	{attribute 'TcIecLibraryType'}
	{attribute 'external_name' := 'F_VN_SeparableCustomFilter_GUID_FC6321D5_149B_44BA_FE2A_AFF910B64319'}
	(* Apply a separable custom filter to the image. *)
	FUNCTION F_VN_SeparableCustomFilter : HRESULT
	VAR_INPUT
		ipSrcImage	:	ITcVnImage;	(* Source image *)
		ipDestImage	:	REFERENCE TO ITcVnImage;	(* Destination image (An appropriate destination image will be created if required.) *)
		eDestDepth	:	ETcVnElementType;	(* Destination image depth *)
	END_VAR
	VAR_IN_OUT
		stKernelX	:	TcVnMatrix;	(* 1D custom row-filter kernel with values of type REAL or LREAL *)
		stKernelY	:	TcVnMatrix;	(* 1D custom column-filter kernel with values of type REAL or LREAL *)
	END_VAR
	VAR_INPUT
		hrPrev	:	HRESULT;	(* HRESULT indicating the result of previous operations (If SUCCEEDED(hrPrev) equals false, no operation is executed.) *)
	END_VAR

END_FUNCTION

// Functions/Image Filtering/F_VN_SeparableCustomFilterExp

	{attribute 'TcIecLibraryType'}
	{attribute 'external_name' := 'F_VN_SeparableCustomFilterExp_GUID_53B70F4F_154A_462E_D532_DBD6B183CFE7'}
	(* Apply a separable custom filter to the image. (expert function) *)
	FUNCTION F_VN_SeparableCustomFilterExp : HRESULT
	VAR_INPUT
		ipSrcImage	:	ITcVnImage;	(* Source image *)
		ipDestImage	:	REFERENCE TO ITcVnImage;	(* Destination image (An appropriate destination image will be created if required.) *)
		eDestDepth	:	ETcVnElementType;	(* Destination image depth *)
	END_VAR
	VAR_IN_OUT
		stKernelX	:	TcVnMatrix;	(* 1D custom row-filter kernel with values of type REAL or LREAL *)
		stKernelY	:	TcVnMatrix;	(* 1D custom column-filter kernel with values of type REAL or LREAL *)
		aAnchor	:	TcVnPoint;	(* Anchor point of the kernel *)
	END_VAR
	VAR_INPUT
		fDelta	:	LREAL;	(* Value added to each pixel after filtering *)
		eBorderType	:	ETcVnBorderInterpolationMethod;	(* Image border handling *)
		hrPrev	:	HRESULT;	(* HRESULT indicating the result of previous operations (If SUCCEEDED(hrPrev) equals false, no operation is executed.) *)
	END_VAR

END_FUNCTION

// Functions/Image Filtering/F_VN_SobelFilter

	{attribute 'TcIecLibraryType'}
	{attribute 'external_name' := 'F_VN_SobelFilter_GUID_E75A9F88_EB52_4C01_DC1F_4C53F4C1A62C'}
	(* Calculates the first, second, or mixed image derivatives using an extended Sobel filter. *)
	FUNCTION F_VN_SobelFilter : HRESULT
	VAR_INPUT
		ipSrcImage	:	ITcVnImage;	(* Source image *)
		ipDestImage	:	REFERENCE TO ITcVnImage;	(* Destination image (An appropriate destination image will be created if required.) *)
		eDestDepth	:	ETcVnElementType;	(* Destination image depth *)
		nXOrder	:	UDINT;	(* Order of the x-derivative (0, 1, 2) *)
		nYOrder	:	UDINT;	(* Order of the y-derivative (0, 1, 2) *)
		hrPrev	:	HRESULT;	(* HRESULT indicating the result of previous operations (If SUCCEEDED(hrPrev) equals false, no operation is executed.) *)
	END_VAR

END_FUNCTION

// Functions/Image Filtering/F_VN_SobelFilterExp

	{attribute 'TcIecLibraryType'}
	{attribute 'external_name' := 'F_VN_SobelFilterExp_GUID_6432B4D4_802B_419E_F701_7BF4156B289B'}
	(* Calculates the first, second, third, or mixed image derivatives using an extended Sobel filter. (expert function) *)
	FUNCTION F_VN_SobelFilterExp : HRESULT
	VAR_INPUT
		ipSrcImage	:	ITcVnImage;	(* Source image *)
		ipDestImage	:	REFERENCE TO ITcVnImage;	(* Destination image (An appropriate destination image will be created if required.) *)
		eDestDepth	:	ETcVnElementType;	(* Destination image depth *)
		nXOrder	:	UDINT;	(* Order of the x-derivative (must be < nKernelSize) *)
		nYOrder	:	UDINT;	(* Order of the y-derivative (must be < nKernelSize) *)
		nKernelSize	:	UDINT;	(* Size of the extended Sobel kernel (3, 5, 7, ..., 31) *)
		fScale	:	LREAL;	(* Scale factor for the computed derivative values *)
		fDelta	:	LREAL;	(* Delta value that is added to the results prior to storing them in dest *)
		eBorderType	:	ETcVnBorderInterpolationMethod;	(* Image border handling *)
		hrPrev	:	HRESULT;	(* HRESULT indicating the result of previous operations (If SUCCEEDED(hrPrev) equals false, no operation is executed.) *)
	END_VAR

END_FUNCTION

// Functions/Image Filtering/F_VN_VarianceFilter

	{attribute 'TcIecLibraryType'}
	{attribute 'external_name' := 'F_VN_VarianceFilter_GUID_EDB0D6CF_7F73_4B27_CF92_1DD3947C3E57'}
	(* Calculates the local variance of an image. *)
	FUNCTION F_VN_VarianceFilter : HRESULT
	VAR_INPUT
		ipSrcImage	:	ITcVnImage;	(* Source image. Only TCVN_ET_USINT Type is supported.  *)
		ipDestImage	:	REFERENCE TO ITcVnImage;	(* Destination image of type TCVN_ET_UINT (An appropriate destination image will be created if required.) *)
		nKernelSize	:	UDINT;	(* Size of the kernel *)
		hrPrev	:	HRESULT;	(* HRESULT indicating the result of previous operations (If SUCCEEDED(hrPrev) equals false, no operation is executed.) *)
	END_VAR

END_FUNCTION

// Functions/Image Filtering/F_VN_VarianceFilterExp

	{attribute 'TcIecLibraryType'}
	{attribute 'external_name' := 'F_VN_VarianceFilterExp_GUID_A7B8D649_AD30_4302_EB39_E9340C7CCFE8'}
	(* Calculates the local variance of an image. (expert function) *)
	FUNCTION F_VN_VarianceFilterExp : HRESULT
	VAR_INPUT
		ipSrcImage	:	ITcVnImage;	(* Source image. Only TCVN_ET_USINT Type is supported. *)
		ipDestImage	:	REFERENCE TO ITcVnImage;	(* Destination image of type TCVN_ET_UINT (An appropriate destination image will be created if required.) *)
		nKernelSize	:	UDINT;	(* Size of the kernel *)
		fScale	:	LREAL;	(* Scale factor for the computed variance values *)
		eBorderType	:	ETcVnBorderInterpolationMethod;	(* Image border handling *)
		hrPrev	:	HRESULT;	(* HRESULT indicating the result of previous operations (If SUCCEEDED(hrPrev) equals false, no operation is executed.) *)
	END_VAR

END_FUNCTION

// Functions/Miscellaneous/F_VN_CheckFunctionInitialization

	{attribute 'TcIecLibraryType'}
	{attribute 'external_name' := 'F_VN_CheckFunctionInitialization_GUID_C3F1DDC0_B6F9_4195_C99F_AF034AC9584D'}
	(* Check if a function is initialized with the specified options. *)
	FUNCTION F_VN_CheckFunctionInitialization : HRESULT
	VAR_INPUT
		eFunction	:	ETcVnInitializableFunction;	(* Initializable function *)
		nOptions	:	ULINT;	(* Initialization options for the function *)
		hrPrev	:	HRESULT;	(* HRESULT indicating the result of previous operations (If SUCCEEDED(hrPrev) equals false, no operation is executed.) *)
	END_VAR

END_FUNCTION

// Functions/Miscellaneous/F_VN_ClipLineToBoundary

	{attribute 'TcIecLibraryType'}
	{attribute 'external_name' := 'F_VN_ClipLineToBoundary_GUID_5BF147CC_4437_4411_DA65_9BE106D06E3D'}
	(* Clips a line to a rectangular boundary. *)
	FUNCTION F_VN_ClipLineToBoundary : HRESULT
	VAR_IN_OUT
		aLine	:	TcVnVector4_LREAL;	(* The first and second element describe the x and y component of the direction vector. The third and fourth element describe the x and y component of the position vector. *)
	END_VAR
	VAR_INPUT
		nX1	:	DINT;	(* x of top left rectangle point *)
		nY1	:	DINT;	(* y of top left rectangle point *)
		nX2	:	DINT;	(* x of bottom right rectangle point *)
		nY2	:	DINT;	(* Y of bottom right rectangle point *)
	END_VAR
	VAR_IN_OUT
		aStartPoint	:	TcVnPoint2_REAL;	(* Returns the clipped starting point of the line. *)
		aEndPoint	:	TcVnPoint2_REAL;	(* Returns the clipped end point of the line. *)
	END_VAR
	VAR_INPUT
		hrPrev	:	HRESULT;	(* HRESULT indicating the result of previous operations (If SUCCEEDED(hrPrev) equals false, no operation is executed.) *)
	END_VAR

END_FUNCTION

// Functions/Miscellaneous/F_VN_ClipLineToBoundary_ITcVnImage

	{attribute 'TcIecLibraryType'}
	{attribute 'external_name' := 'F_VN_ClipLineToBoundary_ITcVnImage_GUID_E0B9D53C_4691_4392_C0F0_296578E237CB'}
	(* Clips a line to the boundary of an image. *)
	FUNCTION F_VN_ClipLineToBoundary_ITcVnImage : HRESULT
	VAR_IN_OUT
		aLine	:	TcVnVector4_LREAL;	(* The first and second element describe the x and y component of the direction vector. The third and fourth element describe the x and y component of the position vector. *)
	END_VAR
	VAR_INPUT
		ipImage	:	ITcVnImage;	(* Image, from which to derive the boundary *)
	END_VAR
	VAR_IN_OUT
		aStartPoint	:	TcVnPoint2_REAL;	(* Returns the clipped starting point of the line. *)
		aEndPoint	:	TcVnPoint2_REAL;	(* Returns the clipped end point of the line. *)
	END_VAR
	VAR_INPUT
		hrPrev	:	HRESULT;	(* HRESULT indicating the result of previous operations (If SUCCEEDED(hrPrev) equals false, no operation is executed.) *)
	END_VAR

END_FUNCTION

// Functions/Miscellaneous/F_VN_ClipLineToBoundary_TcVnRectangle_DINT

	{attribute 'TcIecLibraryType'}
	{attribute 'external_name' := 'F_VN_ClipLineToBoundary_TcVnRectangle_DINT_GUID_83796845_DAE2_42E1_D405_180DCCA547A8'}
	(* Clips a line to a rectangular boundary. *)
	FUNCTION F_VN_ClipLineToBoundary_TcVnRectangle_DINT : HRESULT
	VAR_IN_OUT
		aLine	:	TcVnVector4_LREAL;	(* The first and second element describe the x and y component of the direction vector. The third and fourth element describe the x and y component of the position vector. *)
		stRectangle	:	TcVnRectangle_DINT;	(* Rectangular boundary *)
		aStartPoint	:	TcVnPoint2_REAL;	(* Returns the clipped starting point of the line. *)
		aEndPoint	:	TcVnPoint2_REAL;	(* Returns the clipped end point of the line. *)
	END_VAR
	VAR_INPUT
		hrPrev	:	HRESULT;	(* HRESULT indicating the result of previous operations (If SUCCEEDED(hrPrev) equals false, no operation is executed.) *)
	END_VAR

END_FUNCTION

// Functions/Miscellaneous/F_VN_ConvertITcUnknownToITcVnBitmapExport

	{attribute 'TcIecLibraryType'}
	{attribute 'external_name' := 'F_VN_ConvertITcUnknownToITcVnBitmapExport_GUID_2ADFAF32_D897_4264_C580_D49D5C531DA7'}
	(* Convert an ITcUnknown interface pointer to an ITcVnBitmapExport interface pointer. The destination pointer will be released (if existing) and set to the source pointer. The source pointer will be set to 0. *)
	FUNCTION F_VN_ConvertITcUnknownToITcVnBitmapExport : HRESULT
	VAR_INPUT
		ipSrc	:	REFERENCE TO ITcUnknown;	(* Source pointer *)
		ipDest	:	REFERENCE TO ITcVnBitmapExport;	(* Destination pointer *)
		hrPrev	:	HRESULT;	(* HRESULT indicating the result of previous operations (If SUCCEEDED(hrPrev) equals false, no operation is executed.) *)
	END_VAR

END_FUNCTION

// Functions/Miscellaneous/F_VN_ConvertITcUnknownToITcVnContainer

	{attribute 'TcIecLibraryType'}
	{attribute 'external_name' := 'F_VN_ConvertITcUnknownToITcVnContainer_GUID_17E3F6C3_BFE3_44EF_FE9F_96A9CAE713C6'}
	(* Convert an ITcUnknown interface pointer to an ITcVnContainer interface pointer. The destination pointer will be released (if existing) and set to the source pointer. The source pointer will be set to 0. *)
	FUNCTION F_VN_ConvertITcUnknownToITcVnContainer : HRESULT
	VAR_INPUT
		ipSrc	:	REFERENCE TO ITcUnknown;	(* Source pointer *)
		ipDest	:	REFERENCE TO ITcVnContainer;	(* Destination pointer *)
		hrPrev	:	HRESULT;	(* HRESULT indicating the result of previous operations (If SUCCEEDED(hrPrev) equals false, no operation is executed.) *)
	END_VAR

END_FUNCTION

// Functions/Miscellaneous/F_VN_ConvertITcUnknownToITcVnImage

	{attribute 'TcIecLibraryType'}
	{attribute 'external_name' := 'F_VN_ConvertITcUnknownToITcVnImage_GUID_181BB9EC_9169_4CB5_D135_A350734A00A3'}
	(* Convert an ITcUnknown interface pointer to an ITcVnImage interface pointer. The destination pointer will be released (if existing) and set to the source pointer. The source pointer will be set to 0. *)
	FUNCTION F_VN_ConvertITcUnknownToITcVnImage : HRESULT
	VAR_INPUT
		ipSrc	:	REFERENCE TO ITcUnknown;	(* Source pointer *)
		ipDest	:	REFERENCE TO ITcVnImage;	(* Destination pointer *)
		hrPrev	:	HRESULT;	(* HRESULT indicating the result of previous operations (If SUCCEEDED(hrPrev) equals false, no operation is executed.) *)
	END_VAR

END_FUNCTION

// Functions/Miscellaneous/F_VN_ConvertITcUnknownToITcVnMlModel

	{attribute 'TcIecLibraryType'}
	{attribute 'external_name' := 'F_VN_ConvertITcUnknownToITcVnMlModel_GUID_04956096_DCE0_4A04_C098_21341EC538B6'}
	(* Convert an ITcUnknown interface pointer to an ITcVnMlModel interface pointer. The destination pointer will be released (if existing) and set to the source pointer. The source pointer will be set to 0. *)
	FUNCTION F_VN_ConvertITcUnknownToITcVnMlModel : HRESULT
	VAR_INPUT
		ipSrc	:	REFERENCE TO ITcUnknown;	(* Source pointer *)
		ipDest	:	REFERENCE TO ITcVnMlModel;	(* Destination pointer *)
		hrPrev	:	HRESULT;	(* HRESULT indicating the result of previous operations (If SUCCEEDED(hrPrev) equals false, no operation is executed.) *)
	END_VAR

END_FUNCTION

// Functions/Miscellaneous/F_VN_DeinitializeFunction

	{attribute 'TcIecLibraryType'}
	{attribute 'external_name' := 'F_VN_DeinitializeFunction_GUID_3E80C87C_FFD6_4472_F925_D1593B2E8057'}
	(* Deinitialize the specified options for the function. *)
	FUNCTION F_VN_DeinitializeFunction : HRESULT
	VAR_INPUT
		eFunction	:	ETcVnInitializableFunction;	(* Initializable function *)
		nOptions	:	ULINT;	(* Initialization options for the function *)
		hrPrev	:	HRESULT;	(* HRESULT indicating the result of previous operations (If SUCCEEDED(hrPrev) equals false, no operation is executed.) *)
	END_VAR

END_FUNCTION

// Functions/Miscellaneous/F_VN_GetTimestamp

	{attribute 'TcIecLibraryType'}
	{attribute 'external_name' := 'F_VN_GetTimestamp_GUID_C21B1878_7687_400A_E2C3_1C9DFD495A93'}
	(* Get the timestamp (actual DC time) from the last change of an object (e.g. ITcVnImage or ITcVnContainer) *)
	FUNCTION F_VN_GetTimestamp : HRESULT
	VAR_INPUT
		ipUnknown	:	ITcUnknown;	(* An object implementing ITcUnknown and ITcVnTimestamp (e.g. ITcVnImage or ITcVnContainer) *)
	END_VAR
	VAR_IN_OUT
		nTimestamp	:	LINT;	(* Returns the timestamp *)
	END_VAR
	VAR_INPUT
		hrPrev	:	HRESULT;	(* HRESULT indicating the result of previous operations (If SUCCEEDED(hrPrev) equals false, no operation is executed.) *)
	END_VAR

END_FUNCTION

// Functions/Miscellaneous/F_VN_HuMomentInvariants

	{attribute 'TcIecLibraryType'}
	{attribute 'external_name' := 'F_VN_HuMomentInvariants_GUID_B8FC2F70_ECC3_4CFA_E257_DA68AE77A56B'}
	(* Computes the Hu moment invariants. *)
	FUNCTION F_VN_HuMomentInvariants : HRESULT
	VAR_IN_OUT
		stMoments	:	TcVnMoments;	(* Moments from which to compute the Hu invariants *)
		aHuInvariants	:	TcVnArray7_LREAL;	(* Returns the Hu moment invariants *)
	END_VAR
	VAR_INPUT
		hrPrev	:	HRESULT;	(* HRESULT indicating the result of previous operations (If SUCCEEDED(hrPrev) equals false, no operation is executed.) *)
	END_VAR

END_FUNCTION

// Functions/Miscellaneous/F_VN_InitMatrixStruct

	{attribute 'TcIecLibraryType'}
	{attribute 'external_name' := 'F_VN_InitMatrixStruct_GUID_83E4EF2C_D846_4DB7_E596_EEDDBE9E95C1'}
	(* Initialize a struct of the type TcVnMatrix extending a buffer with metainformation so that it can be used as a matrix. *)
	FUNCTION F_VN_InitMatrixStruct : HRESULT
	VAR_INPUT
		pSrcBuffer	:	PVOID;	(* Source buffer *)
	END_VAR
	VAR_IN_OUT
		stDestMatrix	:	TcVnMatrix;	(* Returns completed matrix struct *)
	END_VAR
	VAR_INPUT
		nRows	:	UDINT;	(* Matrix rows *)
		nCols	:	UDINT;	(* Matrix columns *)
		eElementType	:	ETcVnElementType;	(* Type of the matrix elements *)
		hrPrev	:	HRESULT;	(* HRESULT indicating the result of previous operations (If SUCCEEDED(hrPrev) equals false, no operation is executed.) *)
	END_VAR

END_FUNCTION

// Functions/Miscellaneous/F_VN_InvertMatrix3x3

	{attribute 'TcIecLibraryType'}
	{attribute 'external_name' := 'F_VN_InvertMatrix3x3_GUID_ECDDE1A7_E1A4_4A8E_DD19_43C6A5A13520'}
	(* Invert a 3x3 matrix. *)
	FUNCTION F_VN_InvertMatrix3x3 : HRESULT
	VAR_IN_OUT
		aSrcMatrix	:	TcVnMatrix3x3_LREAL;	(* Source matrix *)
		aInvertedMatrix	:	TcVnMatrix3x3_LREAL;	(* Returns inverted matrix *)
	END_VAR
	VAR_INPUT
		hrPrev	:	HRESULT;	(* HRESULT indicating the result of previous operations (If SUCCEEDED(hrPrev) equals false, no operation is executed.) *)
	END_VAR

END_FUNCTION

// Functions/Miscellaneous/F_VN_LineIntersectionPoint

	{attribute 'TcIecLibraryType'}
	{attribute 'external_name' := 'F_VN_LineIntersectionPoint_GUID_0DB2487D_C450_497D_EABE_6918FECA9855'}
	(* Computes the intersection point between two lines (returns S_FALSE if the provided lines are parallel). *)
	FUNCTION F_VN_LineIntersectionPoint : HRESULT
	VAR_IN_OUT
		aLine1	:	TcVnVector4_LREAL;	(* First line. The first and second element describe the x and y component of a vector collinear to the line. The third and fourth element describe the x and y component of a point on the line. *)
		aLine2	:	TcVnVector4_LREAL;	(* Second line. The first and second element describe the x and y component of a vector collinear to the line. The third and fourth element describe the x and y component of a point on the line. *)
		aIntersecPoint	:	TcVnPoint2_REAL;	(* Returns the intersection point of aLine1 and aLine2. *)
	END_VAR
	VAR_INPUT
		hrPrev	:	HRESULT;	(* HRESULT indicating the result of previous operations (If SUCCEEDED(hrPrev) equals false, no operation is executed.) *)
	END_VAR

END_FUNCTION

// Functions/Miscellaneous/F_VN_LineIntersectionPointAndAngle

	{attribute 'TcIecLibraryType'}
	{attribute 'external_name' := 'F_VN_LineIntersectionPointAndAngle_GUID_06C0B65B_BEEF_48A8_ED9F_979E899E4C6C'}
	(* Computes the intersection point and angle between two lines (returns S_FALSE if the provided lines are parallel). *)
	FUNCTION F_VN_LineIntersectionPointAndAngle : HRESULT
	VAR_IN_OUT
		aLine1	:	TcVnVector4_LREAL;	(* First line. The first and second element describe the x and y component of a vector collinear to the line. The third and fourth element describe the x and y component of a point on the line. *)
		aLine2	:	TcVnVector4_LREAL;	(* Second line. The first and second element describe the x and y component of a vector collinear to the line. The third and fourth element describe the x and y component of a point on the line. *)
		aIntersecPoint	:	TcVnPoint2_REAL;	(* Returns the intersection point of aLine1 and aLine2. *)
		fAngle	:	REAL;	(* Returns the intersection angle of aLine1 and aLine2. *)
	END_VAR
	VAR_INPUT
		bAngleInDegrees	:	BOOL;	(* If TRUE, fAngle is in degrees. If FALSE, fAngle is in radians. *)
		hrPrev	:	HRESULT;	(* HRESULT indicating the result of previous operations (If SUCCEEDED(hrPrev) equals false, no operation is executed.) *)
	END_VAR

END_FUNCTION

// Functions/Miscellaneous/F_VN_MultiplyMatrices

	{attribute 'TcIecLibraryType'}
	{attribute 'external_name' := 'F_VN_MultiplyMatrices_GUID_EA37B7A4_D1DF_4AB1_E9C9_495990E4F4E9'}
	(* Matrix multiplication of two matrices (A * B = C). All matrices are represented by structs holding a pointer to an array of the appropriate size. *)
	FUNCTION F_VN_MultiplyMatrices : HRESULT
	VAR_IN_OUT
		stSrcMatrix1	:	TcVnMatrix;	(* First source matrix (A) *)
		stSrcMatrix2	:	TcVnMatrix;	(* Second source matrix (B) *)
		stDestMatrix	:	TcVnMatrix;	(* Destination matrix (C) (The destination matrix is filled by this function, but the required memory needs to be provided.) *)
	END_VAR
	VAR_INPUT
		hrPrev	:	HRESULT;	(* HRESULT indicating the result of previous operations (If SUCCEEDED(hrPrev) equals false, no operation is executed.) *)
	END_VAR

END_FUNCTION

// Functions/Miscellaneous/F_VN_RotatedRectangleCorners

	{attribute 'TcIecLibraryType'}
	{attribute 'external_name' := 'F_VN_RotatedRectangleCorners_GUID_365D89A9_58B4_4A5A_F2FF_B1BCBFB2313D'}
	(* Computes the 4 corner points of a rotated rectangle. *)
	FUNCTION F_VN_RotatedRectangleCorners : HRESULT
	VAR_IN_OUT
		stRect	:	TcVnRotatedRectangle;	(* Rotated rectangle *)
		aCorners	:	TcVnArray4_Point2_REAL;	(* Returns the 4 corner points *)
	END_VAR
	VAR_INPUT
		hrPrev	:	HRESULT;	(* HRESULT indicating the result of previous operations (If SUCCEEDED(hrPrev) equals false, no operation is executed.) *)
	END_VAR

END_FUNCTION

// Functions/Miscellaneous/F_VN_RotatedRectangleIntersection

	{attribute 'TcIecLibraryType'}
	{attribute 'external_name' := 'F_VN_RotatedRectangleIntersection_GUID_9B131643_76C8_46C1_F46A_E0891B2EA52B'}
	(* Finds the intersection of 2 rotated rectangles. *)
	FUNCTION F_VN_RotatedRectangleIntersection : HRESULT
	VAR_IN_OUT
		stRect1	:	TcVnRotatedRectangle;	(* Rotated rectangle 1 *)
		stRect2	:	TcVnRotatedRectangle;	(* Rotated rectangle 2 *)
	END_VAR
	VAR_INPUT
		ipIntersection	:	REFERENCE TO ITcVnContainer;	(* Returns the intersection points (ContainerType_Vector_TcVnPoint2_REAL, non-zero interface pointers are reused) *)
	END_VAR
	VAR_IN_OUT
		eIntersection	:	ETcVnRectangleIntersection;	(* Returns the intersection type *)
	END_VAR
	VAR_INPUT
		hrPrev	:	HRESULT;	(* HRESULT indicating the result of previous operations (If SUCCEEDED(hrPrev) equals false, no operation is executed.) *)
	END_VAR

END_FUNCTION

// Functions/Miscellaneous/F_VN_SetRngSeed

	{attribute 'TcIecLibraryType'}
	{attribute 'external_name' := 'F_VN_SetRngSeed_GUID_8DE1ABF6_AF04_45F2_FC57_62569F5F6E0B'}
	(* Sets the internal pseudo random number generator seed (intended for testing purposes only). *)
	FUNCTION F_VN_SetRngSeed : HRESULT
	VAR_INPUT
		nSeed	:	DINT;	(* seed (0 sets the generator back to its initial state) *)
		hrPrev	:	HRESULT;	(* HRESULT indicating the result of previous operations (If SUCCEEDED(hrPrev) equals false, no operation is executed.) *)
	END_VAR

END_FUNCTION

// Functions/Miscellaneous/F_VN_UpdateTimestamp

	{attribute 'TcIecLibraryType'}
	{attribute 'external_name' := 'F_VN_UpdateTimestamp_GUID_5BCDAFED_7DEA_4AA0_CDAE_2780A09F469E'}
	(* Update the timestamp of an object to the actual DC time (e.g. ITcVnImage or ITcVnContainer) *)
	FUNCTION F_VN_UpdateTimestamp : HRESULT
	VAR_INPUT
		ipUnknown	:	ITcUnknown;	(* An object implementing ITcUnknown and ITcVnTimestamp (e.g. ITcVnImage or ITcVnContainer) *)
		hrPrev	:	HRESULT;	(* HRESULT indicating the result of previous operations (If SUCCEEDED(hrPrev) equals false, no operation is executed.) *)
	END_VAR

END_FUNCTION

// Functions/Basic Image Operations/F_VN_CombineImageChannels

	{attribute 'TcIecLibraryType'}
	{attribute 'external_name' := 'F_VN_CombineImageChannels_GUID_CAA9C562_D9D6_469F_F6BF_DAE2BF9823AC'}
	(* Combines several single-channel images into one multi-channel image. *)
	FUNCTION F_VN_CombineImageChannels : HRESULT
	VAR_INPUT
		pSrcImages	:	PVOID;	(* Pointer to an array of single-channel source images *)
		ipDestImage	:	REFERENCE TO ITcVnImage;	(* Multi-channel destination image (An appropriate destination image will be created if required.) *)
		nSrcArraySize	:	UINT;	(* pSrcImages array size *)
		hrPrev	:	HRESULT;	(* HRESULT indicating the result of previous operations (If SUCCEEDED(hrPrev) equals false, no operation is executed.) *)
	END_VAR

END_FUNCTION

// Functions/Basic Image Operations/F_VN_ConvertElementType

	{attribute 'TcIecLibraryType'}
	{attribute 'external_name' := 'F_VN_ConvertElementType_GUID_6B133E81_369F_4F2F_DD06_8099166993C8'}
	(* Converts an image to another element type. *)
	FUNCTION F_VN_ConvertElementType : HRESULT
	VAR_INPUT
		ipSrcImage	:	ITcVnImage;	(* Source image *)
		ipDestImage	:	REFERENCE TO ITcVnImage;	(* Destination image (An appropriate destination image will be created if required.) *)
		eElementType	:	ETcVnElementType;	(* Desired element type of the destination image *)
		hrPrev	:	HRESULT;	(* HRESULT indicating the result of previous operations (If SUCCEEDED(hrPrev) equals false, no operation is executed.) *)
	END_VAR

END_FUNCTION

// Functions/Basic Image Operations/F_VN_ConvertElementTypeExp

	{attribute 'TcIecLibraryType'}
	{attribute 'external_name' := 'F_VN_ConvertElementTypeExp_GUID_9BE4A1AB_57F3_43D2_C41F_9A9B55758F93'}
	(* Converts an image to another element type. (expert function) *)
	FUNCTION F_VN_ConvertElementTypeExp : HRESULT
	VAR_INPUT
		ipSrcImage	:	ITcVnImage;	(* Source image *)
		ipDestImage	:	REFERENCE TO ITcVnImage;	(* Destination image (An appropriate destination image will be created if required.) *)
		eElementType	:	ETcVnElementType;	(* Desired element type of the destination image *)
		fScaleFactor	:	LREAL;	(* Scale factor for the pixel values *)
		fDelta	:	LREAL;	(* Value that is added to the scaled pixel values *)
		hrPrev	:	HRESULT;	(* HRESULT indicating the result of previous operations (If SUCCEEDED(hrPrev) equals false, no operation is executed.) *)
	END_VAR

END_FUNCTION

// Functions/Basic Image Operations/F_VN_CopyImage

	{attribute 'TcIecLibraryType'}
	{attribute 'external_name' := 'F_VN_CopyImage_GUID_35BCD2D0_6126_465D_EECE_FD2EE9AC9850'}
	(* Creates a deep copy of an image. *)
	FUNCTION F_VN_CopyImage : HRESULT
	VAR_INPUT
		ipSrcImage	:	ITcVnImage;	(* Source image *)
		ipDestImage	:	REFERENCE TO ITcVnImage;	(* Destination image (An appropriate destination image will be created if required.) *)
		hrPrev	:	HRESULT;	(* HRESULT indicating the result of previous operations (If SUCCEEDED(hrPrev) equals false, no operation is executed.) *)
	END_VAR

END_FUNCTION

// Functions/Basic Image Operations/F_VN_CopyImageRegion

	{attribute 'TcIecLibraryType'}
	{attribute 'external_name' := 'F_VN_CopyImageRegion_GUID_0C8CB38B_7E33_4481_DD06_1AABA6722DFF'}
	(* Deep copy the specified region of interest into a new image. *)
	FUNCTION F_VN_CopyImageRegion : HRESULT
	VAR_INPUT
		ipSrcImage	:	ITcVnImage;	(* Source image *)
		nX	:	UDINT;	(* Left boundary (inclusive 0-based index) *)
		nY	:	UDINT;	(* Upper boundary (inclusive 0-based index) *)
		nWidth	:	UDINT;	(* ROI width *)
		nHeight	:	UDINT;	(* ROI height *)
		ipDestImage	:	REFERENCE TO ITcVnImage;	(* Destination image (An appropriate destination image will be created if required.) *)
		hrPrev	:	HRESULT;	(* HRESULT indicating the result of previous operations (If SUCCEEDED(hrPrev) equals false, no operation is executed.) *)
	END_VAR

END_FUNCTION

// Functions/Basic Image Operations/F_VN_CopyImageRegionToRegion

	{attribute 'TcIecLibraryType'}
	{attribute 'external_name' := 'F_VN_CopyImageRegionToRegion_GUID_9BA3BE0F_2298_4630_F725_091D59484D85'}
	(* Copy an image region into another image region. *)
	FUNCTION F_VN_CopyImageRegionToRegion : HRESULT
	VAR_INPUT
		ipSrcImage	:	ITcVnImage;	(* Source image *)
		nXSrc	:	UDINT;	(* Left boundary in ipSrcImage (inclusive 0-based index) *)
		nYSrc	:	UDINT;	(* Upper boundary in ipSrcImage (inclusive 0-based index) *)
		nWidth	:	UDINT;	(* ROI width *)
		nHeight	:	UDINT;	(* ROI height *)
		ipDestImage	:	ITcVnImage;	(* Destination image (same type as ipSrcImage) *)
		nXDest	:	UDINT;	(* Left boundary in ipDestImage (inclusive 0-based index) *)
		nYDest	:	UDINT;	(* Upper boundary in ipDestImage (inclusive 0-based index) *)
		hrPrev	:	HRESULT;	(* HRESULT indicating the result of previous operations (If SUCCEEDED(hrPrev) equals false, no operation is executed.) *)
	END_VAR

END_FUNCTION

// Functions/Basic Image Operations/F_VN_CopyIntoDisplayableImage

	{attribute 'TcIecLibraryType'}
	{attribute 'external_name' := 'F_VN_CopyIntoDisplayableImage_GUID_9F369AFC_132B_4503_EBE0_B18E5B2854E9'}
	(* Copys an image into a displayable image. If you do not want to use ipSrcImage after this function call, you might want to use F_VN_TransformIntoDisplayableImage instead for better performance. *)
	FUNCTION F_VN_CopyIntoDisplayableImage : HRESULT
	VAR_INPUT
		ipSrcImage	:	ITcVnImage;	(* Source image *)
		ipDestImage	:	REFERENCE TO ITcVnDisplayableImage;	(* Returns the displayable image *)
		hrPrev	:	HRESULT;	(* HRESULT indicating the result of previous operations (If SUCCEEDED(hrPrev) equals false, no operation is executed.) *)
	END_VAR

END_FUNCTION

// Functions/Basic Image Operations/F_VN_TransformIntoDisplayableImage

	{attribute 'TcIecLibraryType'}
	{attribute 'external_name' := 'F_VN_TransformIntoDisplayableImage_GUID_6EB802F3_4901_4623_FC8E_CEF0C004525C'}
	(* Transform an image into a displayable image. The source image will be released and zeroed while existing destination images will be released and overwritten with the function result. The source image must not be used anywhere else and the transformation is very fast. If you want to use ipSrcImage after this function call, use F_VN_CopyIntoDisplayableImage instead. *)
	FUNCTION F_VN_TransformIntoDisplayableImage : HRESULT
	VAR_INPUT
		ipSrcImage	:	REFERENCE TO ITcVnImage;	(* Source image *)
		ipDestImage	:	REFERENCE TO ITcVnDisplayableImage;	(* Returns the displayable image *)
		hrPrev	:	HRESULT;	(* HRESULT indicating the result of previous operations (If SUCCEEDED(hrPrev) equals false, no operation is executed.) *)
	END_VAR

END_FUNCTION

// Functions/Basic Image Operations/F_VN_CreateAssociatedImage

	{attribute 'TcIecLibraryType'}
	{attribute 'external_name' := 'F_VN_CreateAssociatedImage_GUID_2C8B501B_A961_4761_C9C7_AA2D3A369F77'}
	(* Creates a new image that shares its data with the source image. E.g. useful to work on different (disjoint) ROIs in parallel. *)
	FUNCTION F_VN_CreateAssociatedImage : HRESULT
	VAR_INPUT
		ipSrcImage	:	ITcVnImage;	(* Source image *)
		ipDestImage	:	REFERENCE TO ITcVnImage;	(* Returns the created image (Non-zero interface pointers are reused.) *)
		hrPrev	:	HRESULT;	(* HRESULT indicating the result of previous operations (If SUCCEEDED(hrPrev) equals false, no operation is executed.) *)
	END_VAR

END_FUNCTION

// Functions/Basic Image Operations/F_VN_CreateEmptyImage

	{attribute 'TcIecLibraryType'}
	{attribute 'external_name' := 'F_VN_CreateEmptyImage_GUID_EB86C5AC_28E8_4710_F6E0_4D4B6E72F004'}
	(* Creates an empty image without allocating any data buffer. The initial reference count is set to one if a new image interface is created and kept, otherwise. *)
	FUNCTION F_VN_CreateEmptyImage : HRESULT
	VAR_INPUT
		ipImage	:	REFERENCE TO ITcVnImage;	(* Returns the created image *)
		hrPrev	:	HRESULT;	(* HRESULT indicating the result of previous operations (If SUCCEEDED(hrPrev) equals false, no operation is executed.) *)
	END_VAR

END_FUNCTION

// Functions/Basic Image Operations/F_VN_CreateImage

	{attribute 'TcIecLibraryType'}
	{attribute 'external_name' := 'F_VN_CreateImage_GUID_E12CC266_EAB8_4FF0_C09F_C5578D0AF87F'}
	(* Creates an image and allocate an appropriate data buffer. The initial reference count is set to one if a new image interface is created and kept, otherwise. *)
	FUNCTION F_VN_CreateImage : HRESULT
	VAR_INPUT
		ipImage	:	REFERENCE TO ITcVnImage;	(* Returns the created image (Non-zero interface pointers are reused.) *)
		nWidth	:	UDINT;	(* Image width *)
		nHeight	:	UDINT;	(* Image height *)
		ePixelType	:	ETcVnElementType;	(* Pixel type *)
		nChannelNum	:	UDINT;	(* Number of channels (1 to 255) *)
		hrPrev	:	HRESULT;	(* HRESULT indicating the result of previous operations (If SUCCEEDED(hrPrev) equals false, no operation is executed.) *)
	END_VAR

END_FUNCTION

// Functions/Basic Image Operations/F_VN_CreateImageAndSetPixels

	{attribute 'TcIecLibraryType'}
	{attribute 'external_name' := 'F_VN_CreateImageAndSetPixels_GUID_C4CAED43_0A1E_46FF_C10D_853FF9B77DB6'}
	(* Creates an image, allocates an appropriate data buffer and sets all pixels to the specified value. The initial reference count is set to one if a new image interface is created and kept, otherwise. *)
	FUNCTION F_VN_CreateImageAndSetPixels : HRESULT
	VAR_INPUT
		ipImage	:	REFERENCE TO ITcVnImage;	(* Returns the created image (Non-zero interface pointers are reused.) *)
		nWidth	:	UDINT;	(* Image width *)
		nHeight	:	UDINT;	(* Image height *)
		ePixelType	:	ETcVnElementType;	(* Pixel type *)
		nChannelNum	:	UDINT;	(* Number of channels (1 to 4) *)
	END_VAR
	VAR_IN_OUT
		aValue	:	TcVnVector4_LREAL;	(* Pixel value *)
	END_VAR
	VAR_INPUT
		hrPrev	:	HRESULT;	(* HRESULT indicating the result of previous operations (If SUCCEEDED(hrPrev) equals false, no operation is executed.) *)
	END_VAR

END_FUNCTION

// Functions/Basic Image Operations/F_VN_CreateImageFromArray

	{attribute 'TcIecLibraryType'}
	{attribute 'external_name' := 'F_VN_CreateImageFromArray_GUID_0D953F85_948E_4A95_C0A8_092D43EDD419'}
	(* Creates an image and initialize it with the provided data. The initial reference count is set to one if a new image interface is created and kept, otherwise. *)
	FUNCTION F_VN_CreateImageFromArray : HRESULT
	VAR_INPUT
		pData	:	PVOID;	(* Pointer to the 1D data array. Make sure that the array contains at least nWidth * nHeight * nChannelNum elements and that the array element type matches ePixelType. *)
		ipImage	:	REFERENCE TO ITcVnImage;	(* Returns the created image (Non-zero interface pointers are reused.) *)
		nWidth	:	UDINT;	(* Image width *)
		nHeight	:	UDINT;	(* Image height *)
		ePixelType	:	ETcVnElementType;	(* Pixel type *)
		nChannelNum	:	UDINT;	(* Number of channels (1 to 255) *)
		hrPrev	:	HRESULT;	(* HRESULT indicating the result of previous operations (If SUCCEEDED(hrPrev) equals false, no operation is executed.) *)
	END_VAR

END_FUNCTION

// Functions/Basic Image Operations/F_VN_ExportImage

	{attribute 'TcIecLibraryType'}
	{attribute 'external_name' := 'F_VN_ExportImage_GUID_7ECB9C10_8164_43F7_CB27_42EDF9F64B4A'}
	(* Exports the image data into a given buffer (e.g. an array). F_VN_ExportImageSize should be called before to get the required buffer size. *)
	FUNCTION F_VN_ExportImage : HRESULT
	VAR_INPUT
		ipImage	:	ITcVnImage;	(* Image *)
		pBuffer	:	PVOID;	(* Pointer to a buffer to store the image data (Make sure to allocate enough memory! The required size in bytes can be determined using the function F_VN_ExportImageSize) *)
		nBufferSize	:	ULINT;	(* Size of the buffer memory in bytes *)
		hrPrev	:	HRESULT;	(* HRESULT indicating the result of previous operations (If SUCCEEDED(hrPrev) equals false, no operation is executed.) *)
	END_VAR

END_FUNCTION

// Functions/Basic Image Operations/F_VN_ExportImageSize

	{attribute 'TcIecLibraryType'}
	{attribute 'external_name' := 'F_VN_ExportImageSize_GUID_F574E2E6_73B3_4CB4_EC45_848392CA1409'}
	(* Get the required buffer size (in bytes) to store the image data. *)
	FUNCTION F_VN_ExportImageSize : HRESULT
	VAR_INPUT
		ipImage	:	ITcVnImage;	(* Image *)
	END_VAR
	VAR_IN_OUT
		nBufferSize	:	ULINT;	(* Returns the required buffer size in bytes *)
	END_VAR
	VAR_INPUT
		hrPrev	:	HRESULT;	(* HRESULT indicating the result of previous operations (If SUCCEEDED(hrPrev) equals false, no operation is executed.) *)
	END_VAR

END_FUNCTION

// Functions/Basic Image Operations/F_VN_ExportImageAsBmp

	{attribute 'TcIecLibraryType'}
	{attribute 'external_name' := 'F_VN_ExportImageAsBmp_GUID_27926B3F_55F0_4D4D_E5E0_FC00ED59D832'}
	(* Exports the image as bitmap into a given buffer (e.g. an array). F_VN_ExportImageAsBmpSize should be called before to get the required buffer size. *)
	FUNCTION F_VN_ExportImageAsBmp : HRESULT
	VAR_INPUT
		ipImage	:	ITcVnImage;	(* Image *)
		pBuffer	:	PVOID;	(* Pointer to a buffer to store the bitmap image (Make sure to allocate enough memory! The required size in bytes can be determined using the function F_VN_ExportImageAsBmpSize) *)
		nBufferSize	:	ULINT;	(* Size of the buffer memory in bytes *)
		hrPrev	:	HRESULT;	(* HRESULT indicating the result of previous operations (If SUCCEEDED(hrPrev) equals false, no operation is executed.) *)
	END_VAR

END_FUNCTION

// Functions/Basic Image Operations/F_VN_ExportImageAsBmpSize

	{attribute 'TcIecLibraryType'}
	{attribute 'external_name' := 'F_VN_ExportImageAsBmpSize_GUID_63811206_5B1A_4020_FFD9_4716AC3EE57E'}
	(* Get the required buffer size (in bytes) to store the image as bitmap. *)
	FUNCTION F_VN_ExportImageAsBmpSize : HRESULT
	VAR_INPUT
		ipImage	:	ITcVnImage;	(* Image *)
	END_VAR
	VAR_IN_OUT
		nBufferSize	:	ULINT;	(* Returns the required buffer size in bytes *)
	END_VAR
	VAR_INPUT
		hrPrev	:	HRESULT;	(* HRESULT indicating the result of previous operations (If SUCCEEDED(hrPrev) equals false, no operation is executed.) *)
	END_VAR

END_FUNCTION

// Functions/Basic Image Operations/F_VN_ExportImageAsBmpExp

	{attribute 'TcIecLibraryType'}
	{attribute 'external_name' := 'F_VN_ExportImageAsBmpExp_GUID_2B2BFF0D_56C4_4410_D63A_9FBB18AA7FA4'}
	(* Exports the image as bitmap into a given buffer (e.g. an array). F_VN_ExportImageAsBmpSizeExp should be called before to get the required buffer size. (expert function) *)
	FUNCTION F_VN_ExportImageAsBmpExp : HRESULT
	VAR_INPUT
		ipImage	:	ITcVnImage;	(* Image *)
		pBuffer	:	PVOID;	(* Pointer to a buffer to store the bitmap image (Make sure to allocate enough memory! The required size in bytes can be determined using the function F_VN_ExportImageAsBmpSizeExp) *)
		nBufferSize	:	ULINT;	(* Size of the buffer memory in bytes *)
		nWidth	:	UDINT;	(* Desired width (or 0 to keep the original width) *)
		nHeight	:	UDINT;	(* Desired height (or 0 to keep the original height) *)
		hrPrev	:	HRESULT;	(* HRESULT indicating the result of previous operations (If SUCCEEDED(hrPrev) equals false, no operation is executed.) *)
	END_VAR

END_FUNCTION

// Functions/Basic Image Operations/F_VN_ExportImageAsBmpSizeExp

	{attribute 'TcIecLibraryType'}
	{attribute 'external_name' := 'F_VN_ExportImageAsBmpSizeExp_GUID_797262C8_950D_4685_EA20_9CDB59D9475A'}
	(* Get the required buffer size (in bytes) to store the image as bitmap. (expert function) *)
	FUNCTION F_VN_ExportImageAsBmpSizeExp : HRESULT
	VAR_INPUT
		ipImage	:	ITcVnImage;	(* Image *)
	END_VAR
	VAR_IN_OUT
		nBufferSize	:	ULINT;	(* Returns the required buffer size in bytes *)
	END_VAR
	VAR_INPUT
		nWidth	:	UDINT;	(* Desired width (or 0 to keep the original width) *)
		nHeight	:	UDINT;	(* Desired height (or 0 to keep the original height) *)
		hrPrev	:	HRESULT;	(* HRESULT indicating the result of previous operations (If SUCCEEDED(hrPrev) equals false, no operation is executed.) *)
	END_VAR

END_FUNCTION

// Functions/Basic Image Operations/F_VN_FuseImages

	{attribute 'TcIecLibraryType'}
	{attribute 'external_name' := 'F_VN_FuseImages_GUID_28AFD428_183B_43A8_F4A5_D3334A6A0638'}
	(* Fuse 2 images vertically (intended for line scan cameras). *)
	FUNCTION F_VN_FuseImages : HRESULT
	VAR_INPUT
		ipSrcImage1	:	ITcVnImage;	(* Source image 1 *)
		ipSrcImage2	:	ITcVnImage;	(* Source image 2 *)
		ipDestImage	:	REFERENCE TO ITcVnImage;	(* Destination image *)
		nFirstLine	:	UDINT;	(* Line index in ipSrcImage1, which is the first line in ipDestImage *)
		nNumLines	:	UDINT;	(* The number of lines that should be copied to ipDestImage, starting with nFirstLine in ipSrcImage1. Once the last line of ipSrcImage1 was copied, the remaining lines are copied from ipSrcImage2, starting at line index 0. *)
		hrPrev	:	HRESULT;	(* HRESULT indicating the result of previous operations (If SUCCEEDED(hrPrev) equals false, no operation is executed.) *)
	END_VAR

END_FUNCTION

// Functions/Basic Image Operations/F_VN_FuseImagesArray

	{attribute 'TcIecLibraryType'}
	{attribute 'external_name' := 'F_VN_FuseImagesArray_GUID_1CA6B3C3_00AA_44A5_F04E_DC07730BD372'}
	(* Fuse up to 10 images vertically (intended for line scan cameras). *)
	FUNCTION F_VN_FuseImagesArray : HRESULT
	VAR_IN_OUT
		aSrcImageArray	:	TcVnArray10_ITcVnImage;	(* Ten-element source image array (not all elements need to be filled, nValidImages specifies the actual amount of images) *)
	END_VAR
	VAR_INPUT
		nValidImages	:	UDINT;	(* Number of valid images in aSrcImageArray *)
		ipDestImage	:	REFERENCE TO ITcVnImage;	(* Destination image *)
		nFirstLine	:	UDINT;	(* Line index in ipSrcImage1, which is the first line in ipDestImage *)
		nNumLines	:	UDINT;	(* The number of lines that should be copied to ipDestImage, starting with nFirstLine in aSrcImageArray[0]. Once the last line of aSrcImageArray[0] was copied, the remaining lines are copied from aSrcImageArray[1] (starting at line index 0) and so on. *)
		hrPrev	:	HRESULT;	(* HRESULT indicating the result of previous operations (If SUCCEEDED(hrPrev) equals false, no operation is executed.) *)
	END_VAR

END_FUNCTION

// Functions/Basic Image Operations/F_VN_GetImageChannel

	{attribute 'TcIecLibraryType'}
	{attribute 'external_name' := 'F_VN_GetImageChannel_GUID_7941C13F_38A1_4023_CDD9_6611D3E36B81'}
	(* Return the specified source image channel as a single-channel image. *)
	FUNCTION F_VN_GetImageChannel : HRESULT
	VAR_INPUT
		ipSrcImage	:	ITcVnImage;	(* Source image *)
		ipDestImage	:	REFERENCE TO ITcVnImage;	(* Destination image (An appropriate image will be created if required.) *)
		nChannelIndex	:	UINT;	(* Index of the requested source image channel *)
		hrPrev	:	HRESULT;	(* HRESULT indicating the result of previous operations (If SUCCEEDED(hrPrev) equals false, no operation is executed.) *)
	END_VAR

END_FUNCTION

// Functions/Basic Image Operations/F_VN_GetImageHeight

	{attribute 'TcIecLibraryType'}
	{attribute 'external_name' := 'F_VN_GetImageHeight_GUID_0987017E_3F8B_434B_C39A_A63D5F3112D9'}
	(* Return the height of an image. (Alternatively use interface method .GetHeight.) *)
	FUNCTION F_VN_GetImageHeight : HRESULT
	VAR_INPUT
		ipImage	:	ITcVnImage;	(* Image *)
	END_VAR
	VAR_IN_OUT
		nHeight	:	UDINT;	(* Return the height of ipImage *)
	END_VAR
	VAR_INPUT
		hrPrev	:	HRESULT;	(* HRESULT indicating the result of previous operations (If SUCCEEDED(hrPrev) equals false, no operation is executed.) *)
	END_VAR

END_FUNCTION

// Functions/Basic Image Operations/F_VN_GetImageInfo

	{attribute 'TcIecLibraryType'}
	{attribute 'external_name' := 'F_VN_GetImageInfo_GUID_48CA8F68_7BEF_44C7_D274_9C74E94FCFAA'}
	(* Gets a struct containing all common meta infos of the image. (Alternatively use interface method .GetImageInfo.) *)
	FUNCTION F_VN_GetImageInfo : HRESULT
	VAR_INPUT
		ipImage	:	ITcVnImage;	(* Image *)
	END_VAR
	VAR_IN_OUT
		stImageInfo	:	TcVnImageInfo;	(* Returns a struct describing the image *)
	END_VAR
	VAR_INPUT
		hrPrev	:	HRESULT;	(* HRESULT indicating the result of previous operations (If SUCCEEDED(hrPrev) equals false, no operation is executed.) *)
	END_VAR

END_FUNCTION

// Functions/Basic Image Operations/F_VN_GetImageWidth

	{attribute 'TcIecLibraryType'}
	{attribute 'external_name' := 'F_VN_GetImageWidth_GUID_3165FD19_0AB9_4F4D_DF4E_3D52DFA18933'}
	(* Return the width of an image. (Alternatively use interface method .GetWidth.) *)
	FUNCTION F_VN_GetImageWidth : HRESULT
	VAR_INPUT
		ipImage	:	ITcVnImage;	(* Image *)
	END_VAR
	VAR_IN_OUT
		nWidth	:	UDINT;	(* Return the width of ipImage *)
	END_VAR
	VAR_INPUT
		hrPrev	:	HRESULT;	(* HRESULT indicating the result of previous operations (If SUCCEEDED(hrPrev) equals false, no operation is executed.) *)
	END_VAR

END_FUNCTION

// Functions/Basic Image Operations/F_VN_GetPixel

	{attribute 'TcIecLibraryType'}
	{attribute 'external_name' := 'F_VN_GetPixel_GUID_338CF121_04E8_452D_C817_86BFF8A99916'}
	(* Gets a specific pixel. *)
	FUNCTION F_VN_GetPixel : HRESULT
	VAR_INPUT
		ipSrcImage	:	ITcVnImage;	(* Source image *)
	END_VAR
	VAR_IN_OUT
		aValue	:	TcVnVector4_LREAL;	(* Returns the pixel value (Unused channels are set to 0.) *)
	END_VAR
	VAR_INPUT
		nX	:	UDINT;	(* x coordinate of the pixel *)
		nY	:	UDINT;	(* y coordinate of the pixel *)
		hrPrev	:	HRESULT;	(* HRESULT indicating the result of previous operations (If SUCCEEDED(hrPrev) equals false, no operation is executed.) *)
	END_VAR

END_FUNCTION

// Functions/Basic Image Operations/F_VN_GetPixelFormat

	{attribute 'TcIecLibraryType'}
	{attribute 'external_name' := 'F_VN_GetPixelFormat_GUID_B884F4D7_289D_42C5_F01F_6CB625E4BF95'}
	(* Gets the pixel format of an image. (Alternatively use interface method .GetPixelFormat.) *)
	FUNCTION F_VN_GetPixelFormat : HRESULT
	VAR_INPUT
		ipImage	:	ITcVnImage;	(* Image *)
	END_VAR
	VAR_IN_OUT
		stPixelFormat	:	TcVnPixelFormat;	(* Returns a struct describing the pixel format *)
	END_VAR
	VAR_INPUT
		hrPrev	:	HRESULT;	(* HRESULT indicating the result of previous operations (If SUCCEEDED(hrPrev) equals false, no operation is executed.) *)
	END_VAR

END_FUNCTION

// Functions/Basic Image Operations/F_VN_GetRoi

	{attribute 'TcIecLibraryType'}
	{attribute 'external_name' := 'F_VN_GetRoi_GUID_7B206172_8208_46C2_CB65_E4E721FE62DF'}
	(* Gets the coordinates of the region of interest (ROI) within the image. *)
	FUNCTION F_VN_GetRoi : HRESULT
	VAR_INPUT
		ipSrcImage	:	ITcVnImage;	(* Source image *)
	END_VAR
	VAR_IN_OUT
		stRoi	:	TcVnRectangle_UDINT;	(* Returns the coordinates of the region of interest *)
	END_VAR
	VAR_INPUT
		hrPrev	:	HRESULT;	(* HRESULT indicating the result of previous operations (If SUCCEEDED(hrPrev) equals false, no operation is executed.) *)
	END_VAR

END_FUNCTION

// Functions/Basic Image Operations/F_VN_MixImageChannels

	{attribute 'TcIecLibraryType'}
	{attribute 'external_name' := 'F_VN_MixImageChannels_GUID_7DA0C6F6_BDF5_4CD2_E97A_6934003070ED'}
	(* Mix image channels by copying the specified channels of the source image into the specified channels of the destination image. *)
	FUNCTION F_VN_MixImageChannels : HRESULT
	VAR_INPUT
		ipSrcImage	:	ITcVnImage;	(* Source image *)
		ipDestImage	:	REFERENCE TO ITcVnImage;	(* Destination image (An appropriate image will be created if required.) *)
		ipIndicesFromTo	:	ITcVnContainer;	(* Index pairs (ContainerType_Vector_TcVnVector2_DINT), specifying which source channel (TcVnVector2_DINT [0]) should be copied to which destination channel (TcVnVector2_DINT [1]). *)
		hrPrev	:	HRESULT;	(* HRESULT indicating the result of previous operations (If SUCCEEDED(hrPrev) equals false, no operation is executed.) *)
	END_VAR

END_FUNCTION

// Functions/Basic Image Operations/F_VN_ResetRoi

	{attribute 'TcIecLibraryType'}
	{attribute 'external_name' := 'F_VN_ResetRoi_GUID_ABB05205_A5DE_4811_D695_A8EFA8D78FDC'}
	(* Reset the region of interest (ROI) of an image. (After this operation, the ROI is set to the entire image.) *)
	FUNCTION F_VN_ResetRoi : HRESULT
	VAR_INPUT
		ipImage	:	ITcVnImage;	(* Image *)
		hrPrev	:	HRESULT;	(* HRESULT indicating the result of previous operations (If SUCCEEDED(hrPrev) equals false, no operation is executed.) *)
	END_VAR

END_FUNCTION

// Functions/Basic Image Operations/F_VN_SetImageChannel

	{attribute 'TcIecLibraryType'}
	{attribute 'external_name' := 'F_VN_SetImageChannel_GUID_8DF17BFC_F855_4131_FEE4_91A604AE4FD9'}
	(* Sets the specified destination image channel to the values of the specified source image channel. *)
	FUNCTION F_VN_SetImageChannel : HRESULT
	VAR_INPUT
		ipSrcImage	:	ITcVnImage;	(* Source image *)
		ipDestImage	:	REFERENCE TO ITcVnImage;	(* Destination image (An appropriate image will be created if required.) *)
		nSrcChannelIndex	:	UINT;	(* Index of the source image channel *)
		nDestChannelIndex	:	UINT;	(* Index of the destination image channel, which will be replaced by the specified source image channel *)
		hrPrev	:	HRESULT;	(* HRESULT indicating the result of previous operations (If SUCCEEDED(hrPrev) equals false, no operation is executed.) *)
	END_VAR

END_FUNCTION

// Functions/Basic Image Operations/F_VN_SetPixel

	{attribute 'TcIecLibraryType'}
	{attribute 'external_name' := 'F_VN_SetPixel_GUID_0CA453E5_A219_456B_D9E2_3AE75CE556EA'}
	(* Sets a specific pixel. *)
	FUNCTION F_VN_SetPixel : HRESULT
	VAR_INPUT
		ipSrcImage	:	ITcVnImage;	(* Source image *)
	END_VAR
	VAR_IN_OUT
		aValue	:	TcVnVector4_LREAL;	(* The pixel value to set (additional channels are ignored.) *)
	END_VAR
	VAR_INPUT
		nX	:	UDINT;	(* x coordinate of the pixel *)
		nY	:	UDINT;	(* y coordinate of the pixel *)
		hrPrev	:	HRESULT;	(* HRESULT indicating the result of previous operations (If SUCCEEDED(hrPrev) equals false, no operation is executed.) *)
	END_VAR

END_FUNCTION

// Functions/Basic Image Operations/F_VN_SetPixels

	{attribute 'TcIecLibraryType'}
	{attribute 'external_name' := 'F_VN_SetPixels_GUID_7D037101_C6C8_4BAF_DF09_20B97DE67DD5'}
	(* Sets all pixels of an image to a given value. *)
	FUNCTION F_VN_SetPixels : HRESULT
	VAR_INPUT
		ipDestImage	:	ITcVnImage;	(* Destination image *)
	END_VAR
	VAR_IN_OUT
		aValue	:	TcVnVector4_LREAL;	(* Pixel value *)
	END_VAR
	VAR_INPUT
		hrPrev	:	HRESULT;	(* HRESULT indicating the result of previous operations (If SUCCEEDED(hrPrev) equals false, no operation is executed.) *)
	END_VAR

END_FUNCTION

// Functions/Basic Image Operations/F_VN_SetPixelsExp

	{attribute 'TcIecLibraryType'}
	{attribute 'external_name' := 'F_VN_SetPixelsExp_GUID_C22B6F4E_E0E5_4703_CB90_D5A1BB64D84F'}
	(* Sets all pixels of an image to a given value. (expert function) *)
	FUNCTION F_VN_SetPixelsExp : HRESULT
	VAR_INPUT
		ipDestImage	:	ITcVnImage;	(* Destination image *)
	END_VAR
	VAR_IN_OUT
		aValue	:	TcVnVector4_LREAL;	(* Pixel value *)
	END_VAR
	VAR_INPUT
		ipMask	:	ITcVnImage;	(* Mask image *)
		hrPrev	:	HRESULT;	(* HRESULT indicating the result of previous operations (If SUCCEEDED(hrPrev) equals false, no operation is executed.) *)
	END_VAR

END_FUNCTION

// Functions/Basic Image Operations/F_VN_SetRoi

	{attribute 'TcIecLibraryType'}
	{attribute 'external_name' := 'F_VN_SetRoi_GUID_ECBFC50B_7037_4170_C30D_137C8CFC25EF'}
	(* Sets a region of interest (ROI) within an image. *)
	FUNCTION F_VN_SetRoi : HRESULT
	VAR_INPUT
		nX	:	UDINT;	(* Left boundary (inclusive 0-based index) *)
		nY	:	UDINT;	(* Upper boundary (inclusive 0-based index) *)
		nWidth	:	UDINT;	(* ROI width *)
		nHeight	:	UDINT;	(* ROI height *)
		ipDestImage	:	ITcVnImage;	(* Destination image *)
		hrPrev	:	HRESULT;	(* HRESULT indicating the result of previous operations (If SUCCEEDED(hrPrev) equals false, no operation is executed.) *)
	END_VAR

END_FUNCTION

// Functions/Basic Image Operations/F_VN_SetRoi_TcVnRectangle_DINT

	{attribute 'TcIecLibraryType'}
	{attribute 'external_name' := 'F_VN_SetRoi_TcVnRectangle_DINT_GUID_B2F48821_2E8B_47BA_DA53_EB95B0025D4C'}
	(* Sets a region of interest (ROI) within an image. *)
	FUNCTION F_VN_SetRoi_TcVnRectangle_DINT : HRESULT
	VAR_IN_OUT
		stRoi	:	TcVnRectangle_DINT;	(* Region of interest *)
	END_VAR
	VAR_INPUT
		ipDestImage	:	ITcVnImage;	(* Destination image *)
		hrPrev	:	HRESULT;	(* HRESULT indicating the result of previous operations (If SUCCEEDED(hrPrev) equals false, no operation is executed.) *)
	END_VAR

END_FUNCTION

// Functions/Basic Image Operations/F_VN_SetRoi_TcVnRectangle_UDINT

	{attribute 'TcIecLibraryType'}
	{attribute 'external_name' := 'F_VN_SetRoi_TcVnRectangle_UDINT_GUID_E7CECB79_85DF_4D0B_DDF0_3AD7FF4D5EDE'}
	(* Sets a region of interest (ROI) within an image. *)
	FUNCTION F_VN_SetRoi_TcVnRectangle_UDINT : HRESULT
	VAR_IN_OUT
		stRoi	:	TcVnRectangle_UDINT;	(* Region of interest *)
	END_VAR
	VAR_INPUT
		ipDestImage	:	ITcVnImage;	(* Destination image *)
		hrPrev	:	HRESULT;	(* HRESULT indicating the result of previous operations (If SUCCEEDED(hrPrev) equals false, no operation is executed.) *)
	END_VAR

END_FUNCTION

// Functions/Basic Image Operations/F_VN_SplitImageChannels

	{attribute 'TcIecLibraryType'}
	{attribute 'external_name' := 'F_VN_SplitImageChannels_GUID_2EBEF070_55AF_4E9E_CF65_B412CF3FA426'}
	(* Split a multi-channel image into multiple single channel images (1 for each source image channel). *)
	FUNCTION F_VN_SplitImageChannels : HRESULT
	VAR_INPUT
		ipSrcImage	:	ITcVnImage;	(* Source image with multiple channels *)
		pDestImages	:	PVOID;	(* Pointer to an array of ITcVnImage (appropriate destination images will be created if required) *)
		nArraySize	:	UINT;	(* Number of pDestImages array elements (array must be >= ipSourceImage channels) *)
		hrPrev	:	HRESULT;	(* HRESULT indicating the result of previous operations (If SUCCEEDED(hrPrev) equals false, no operation is executed.) *)
	END_VAR
	VAR_OUTPUT
		nImageChannels	:	UINT;	(* Actual source image channels *)
	END_VAR

END_FUNCTION

// Functions/Basic Image Operations/F_VN_TransformIntoDisplayableImageExp

	{attribute 'TcIecLibraryType'}
	{attribute 'external_name' := 'F_VN_TransformIntoDisplayableImageExp_GUID_919A3258_B98E_45F7_C551_05F8BB41D851'}
	(* Transform an image into a displayable image. The source image will be released and zeroed while existing destination images will be released and overwritten with the function result. If bAllowDeepCopy equals false, the source image must not be used anywhere else and the transformation is always very fast. Otherwise, if bAllowDeepCopy equals true, a deep copy of the source image might be created if required, which will result in a longer execution time. If you want to use ipSrcImage after this function call, use F_VN_CopyIntoDisplayableImage instead. (expert function) *)
	FUNCTION F_VN_TransformIntoDisplayableImageExp : HRESULT
	VAR_INPUT
		ipSrcImage	:	REFERENCE TO ITcVnImage;	(* Source image *)
		ipDestImage	:	REFERENCE TO ITcVnDisplayableImage;	(* Returns the displayable image *)
		bAllowDeepCopy	:	BOOL;	(* Allow deep image copies, if required *)
		hrPrev	:	HRESULT;	(* HRESULT indicating the result of previous operations (If SUCCEEDED(hrPrev) equals false, no operation is executed.) *)
	END_VAR

END_FUNCTION

// Functions/Container Statistics/F_VN_ContainerAverage

	{attribute 'TcIecLibraryType'}
	{attribute 'external_name' := 'F_VN_ContainerAverage_GUID_2D6890FE_3D5D_45FC_EE16_50733A3EACCC'}
	(* Calculate the average of elements in a container. *)
	FUNCTION F_VN_ContainerAverage : HRESULT
	VAR_INPUT
		ipSrcContainer	:	ITcVnContainer;	(* Source container (Arithmetic, point and vector element types are supported. For points and vectors, the euclidean norm is used.) *)
	END_VAR
	VAR_IN_OUT
		fAverage	:	LREAL;	(* Returns the calculated average value *)
	END_VAR
	VAR_INPUT
		hrPrev	:	HRESULT;	(* HRESULT indicating the result of previous operations (If SUCCEEDED(hrPrev) equals false, no operation is executed.) *)
	END_VAR

END_FUNCTION

// Functions/Container Statistics/F_VN_ContainerAverageElementwise2

	{attribute 'TcIecLibraryType'}
	{attribute 'external_name' := 'F_VN_ContainerAverageElementwise2_GUID_227620A1_EDC4_470B_E7AC_D4453245048E'}
	(* Calculate the elementwise average of 2D elements in a container. *)
	FUNCTION F_VN_ContainerAverageElementwise2 : HRESULT
	VAR_INPUT
		ipSrcContainer	:	ITcVnContainer;	(* Source container with 2D points or vectors *)
	END_VAR
	VAR_IN_OUT
		aAverage	:	TcVnVector2_LREAL;	(* Returns the calculated average values *)
	END_VAR
	VAR_INPUT
		hrPrev	:	HRESULT;	(* HRESULT indicating the result of previous operations (If SUCCEEDED(hrPrev) equals false, no operation is executed.) *)
	END_VAR

END_FUNCTION

// Functions/Container Statistics/F_VN_ContainerAverageElementwise3

	{attribute 'TcIecLibraryType'}
	{attribute 'external_name' := 'F_VN_ContainerAverageElementwise3_GUID_C71EFB8F_E0BD_4D5A_C285_85BEA6DD80EC'}
	(* Calculate the elementwise average of 3D elements in a container. *)
	FUNCTION F_VN_ContainerAverageElementwise3 : HRESULT
	VAR_INPUT
		ipSrcContainer	:	ITcVnContainer;	(* Source container with 3D points or vectors *)
	END_VAR
	VAR_IN_OUT
		aAverage	:	TcVnVector3_LREAL;	(* Returns the calculated average values *)
	END_VAR
	VAR_INPUT
		hrPrev	:	HRESULT;	(* HRESULT indicating the result of previous operations (If SUCCEEDED(hrPrev) equals false, no operation is executed.) *)
	END_VAR

END_FUNCTION

// Functions/Container Statistics/F_VN_ContainerAverageElementwise4

	{attribute 'TcIecLibraryType'}
	{attribute 'external_name' := 'F_VN_ContainerAverageElementwise4_GUID_594C54B5_520C_44AE_EB18_2C1F14EBF18E'}
	(* Calculate the elementwise average of 4D elements in a container. *)
	FUNCTION F_VN_ContainerAverageElementwise4 : HRESULT
	VAR_INPUT
		ipSrcContainer	:	ITcVnContainer;	(* Source container with 4D vectors *)
	END_VAR
	VAR_IN_OUT
		aAverage	:	TcVnVector4_LREAL;	(* Returns the calculated average values *)
	END_VAR
	VAR_INPUT
		hrPrev	:	HRESULT;	(* HRESULT indicating the result of previous operations (If SUCCEEDED(hrPrev) equals false, no operation is executed.) *)
	END_VAR

END_FUNCTION

// Functions/Container Statistics/F_VN_ContainerAverageVariance

	{attribute 'TcIecLibraryType'}
	{attribute 'external_name' := 'F_VN_ContainerAverageVariance_GUID_7F8DFCB4_ADC7_4982_E0E2_F1C10709D26C'}
	(* Calculate the average and variance of elements in a container. *)
	FUNCTION F_VN_ContainerAverageVariance : HRESULT
	VAR_INPUT
		ipSrcContainer	:	ITcVnContainer;	(* Source container (Arithmetic, point and vector element types are supported. For points and vectors, the euclidean norm is used.) *)
	END_VAR
	VAR_IN_OUT
		fAverage	:	LREAL;	(* Returns the calculated average value *)
		fVariance	:	LREAL;	(* Returns the calculated variance value *)
	END_VAR
	VAR_INPUT
		hrPrev	:	HRESULT;	(* HRESULT indicating the result of previous operations (If SUCCEEDED(hrPrev) equals false, no operation is executed.) *)
	END_VAR

END_FUNCTION

// Functions/Container Statistics/F_VN_ContainerAverageVarianceElementwise2

	{attribute 'TcIecLibraryType'}
	{attribute 'external_name' := 'F_VN_ContainerAverageVarianceElementwise2_GUID_1A387EFF_7629_4277_EDBE_8C90D8FADBB5'}
	(* Calculate the elementwise average and variance of 2D elements in a container. *)
	FUNCTION F_VN_ContainerAverageVarianceElementwise2 : HRESULT
	VAR_INPUT
		ipSrcContainer	:	ITcVnContainer;	(* Source container with 2D points or vectors *)
	END_VAR
	VAR_IN_OUT
		aAverage	:	TcVnVector2_LREAL;	(* Returns the calculated average values *)
		aVariance	:	TcVnVector2_LREAL;	(* Returns the calculated variance values *)
	END_VAR
	VAR_INPUT
		hrPrev	:	HRESULT;	(* HRESULT indicating the result of previous operations (If SUCCEEDED(hrPrev) equals false, no operation is executed.) *)
	END_VAR

END_FUNCTION

// Functions/Container Statistics/F_VN_ContainerAverageVarianceElementwise3

	{attribute 'TcIecLibraryType'}
	{attribute 'external_name' := 'F_VN_ContainerAverageVarianceElementwise3_GUID_7D63F050_C65D_4A9A_F822_4116882A3489'}
	(* Calculate the elementwise average and variance of 3D elements in a container. *)
	FUNCTION F_VN_ContainerAverageVarianceElementwise3 : HRESULT
	VAR_INPUT
		ipSrcContainer	:	ITcVnContainer;	(* Source container with 3D points or vectors *)
	END_VAR
	VAR_IN_OUT
		aAverage	:	TcVnVector3_LREAL;	(* Returns the calculated average values *)
		aVariance	:	TcVnVector3_LREAL;	(* Returns the calculated variance values *)
	END_VAR
	VAR_INPUT
		hrPrev	:	HRESULT;	(* HRESULT indicating the result of previous operations (If SUCCEEDED(hrPrev) equals false, no operation is executed.) *)
	END_VAR

END_FUNCTION

// Functions/Container Statistics/F_VN_ContainerAverageVarianceElementwise4

	{attribute 'TcIecLibraryType'}
	{attribute 'external_name' := 'F_VN_ContainerAverageVarianceElementwise4_GUID_84FEB3CC_7438_4443_D19A_1067BD8A2AC5'}
	(* Calculate the elementwise average and variance of 4D elements in a container. *)
	FUNCTION F_VN_ContainerAverageVarianceElementwise4 : HRESULT
	VAR_INPUT
		ipSrcContainer	:	ITcVnContainer;	(* Source container with 4D vectors *)
	END_VAR
	VAR_IN_OUT
		aAverage	:	TcVnVector4_LREAL;	(* Returns the calculated average values *)
		aVariance	:	TcVnVector4_LREAL;	(* Returns the calculated variance values *)
	END_VAR
	VAR_INPUT
		hrPrev	:	HRESULT;	(* HRESULT indicating the result of previous operations (If SUCCEEDED(hrPrev) equals false, no operation is executed.) *)
	END_VAR

END_FUNCTION

// Functions/Container Statistics/F_VN_MaxElement

	{attribute 'TcIecLibraryType'}
	{attribute 'external_name' := 'F_VN_MaxElement_GUID_14B3129F_2FC7_4B61_C1F6_2D636BE355DB'}
	(* Gets the maximum element of a container. *)
	FUNCTION F_VN_MaxElement : HRESULT
	VAR_INPUT
		ipSrcContainer	:	ITcVnContainer;	(* Source container (Arithmetic, point and vector element types are supported. For points and vectors, the euclidean norm is used.) *)
		ipDestIterator	:	REFERENCE TO ITcVnBidirectionalIterator;	(* Returns an iterator to the requested element *)
	END_VAR
	VAR_IN_OUT
		nIndex	:	ULINT;	(* Returns the position of the requested element within the container *)
	END_VAR
	VAR_INPUT
		hrPrev	:	HRESULT;	(* HRESULT indicating the result of previous operations (If SUCCEEDED(hrPrev) equals false, no operation is executed.) *)
	END_VAR

END_FUNCTION

// Functions/Container Statistics/F_VN_MedianElement

	{attribute 'TcIecLibraryType'}
	{attribute 'external_name' := 'F_VN_MedianElement_GUID_F4A6AD1C_3B86_4524_DA8B_8DF6D1C076D2'}
	(* Gets the median element of a container. *)
	FUNCTION F_VN_MedianElement : HRESULT
	VAR_INPUT
		ipSrcContainer	:	ITcVnContainer;	(* Source container (Arithmetic, point and vector element types are supported. For points and vectors, the euclidean norm is used.) *)
		ipDestIterator	:	REFERENCE TO ITcVnBidirectionalIterator;	(* Returns an iterator to the requested element *)
	END_VAR
	VAR_IN_OUT
		nIndex	:	ULINT;	(* Returns the position of the requested element within the container *)
	END_VAR
	VAR_INPUT
		hrPrev	:	HRESULT;	(* HRESULT indicating the result of previous operations (If SUCCEEDED(hrPrev) equals false, no operation is executed.) *)
	END_VAR

END_FUNCTION

// Functions/Container Statistics/F_VN_MinElement

	{attribute 'TcIecLibraryType'}
	{attribute 'external_name' := 'F_VN_MinElement_GUID_12834FFF_2BEA_4951_E5C4_816721F143F5'}
	(* Gets the minimum element of a container. *)
	FUNCTION F_VN_MinElement : HRESULT
	VAR_INPUT
		ipSrcContainer	:	ITcVnContainer;	(* Source container (Arithmetic, point and vector element types are supported. For points and vectors, the euclidean norm is used.) *)
		ipDestIterator	:	REFERENCE TO ITcVnBidirectionalIterator;	(* Returns an iterator to the requested element *)
	END_VAR
	VAR_IN_OUT
		nIndex	:	ULINT;	(* Returns the position of the requested element within the container *)
	END_VAR
	VAR_INPUT
		hrPrev	:	HRESULT;	(* HRESULT indicating the result of previous operations (If SUCCEEDED(hrPrev) equals false, no operation is executed.) *)
	END_VAR

END_FUNCTION

// Functions/Fourier Analysis/F_VN_CreateBandpassButterworthFilter

	{attribute 'TcIecLibraryType'}
	{attribute 'external_name' := 'F_VN_CreateBandpassButterworthFilter_GUID_2391300F_96D6_48F0_E7E7_A10C8921A45D'}
	(* Creates a bandpass Butterworth filter, which can be applied to a frequency domain image by element-wise multiplication. *)
	FUNCTION F_VN_CreateBandpassButterworthFilter : HRESULT
	VAR_INPUT
		ipFilter	:	REFERENCE TO ITcVnImage;	(* Returns the created filter (1 channel of type REAL or LREAL, depending on bDoublePrecision. Non-zero interface pointers are reused.). *)
		nWidth	:	UDINT;	(* Filter width (even, >= 2, must match the width of the image it is applied to) *)
		nHeight	:	UDINT;	(* Filter height (even, >= 2, must match the height of the image it is applied to) *)
		bDoublePrecision	:	BOOL;	(* If true, the filter is generated with double precision (LREAL) instead of single precision (REAL). *)
		bOriginAtCenter	:	BOOL;	(* If true, the filter origin is shifted to the image center. *)
		fCutoffDistance	:	LREAL;	(* The cutoff distance of the Butterworth filter (> 0). *)
		fBandWidth	:	LREAL;	(* The band width of the Butterworth filter (> 0). *)
		nOrder	:	UDINT;	(* The order of the Butterworth filter (> 0). *)
		fScale	:	LREAL;	(* The scale factor of the Butterworth filter denominator term (> 0, e.g. 0.414 or 1.0). *)
		hrPrev	:	HRESULT;	(* HRESULT indicating the result of previous operations (If SUCCEEDED(hrPrev) equals false, no operation is executed.) *)
	END_VAR

END_FUNCTION

// Functions/Fourier Analysis/F_VN_CreateBandpassGaussianFilter

	{attribute 'TcIecLibraryType'}
	{attribute 'external_name' := 'F_VN_CreateBandpassGaussianFilter_GUID_2CDEA4C2_A425_4B8E_D535_B765577363A2'}
	(* Creates a bandpass Gaussian filter, which can be applied to a frequency domain image by element-wise multiplication. *)
	FUNCTION F_VN_CreateBandpassGaussianFilter : HRESULT
	VAR_INPUT
		ipFilter	:	REFERENCE TO ITcVnImage;	(* Returns the created filter (1 channel of type REAL or LREAL, depending on bDoublePrecision. Non-zero interface pointers are reused.). *)
		nWidth	:	UDINT;	(* Filter width (even, >= 2, must match the width of the image it is applied to) *)
		nHeight	:	UDINT;	(* Filter height (even, >= 2, must match the height of the image it is applied to) *)
		bDoublePrecision	:	BOOL;	(* If true, the filter is generated with double precision (LREAL) instead of single precision (REAL). *)
		bOriginAtCenter	:	BOOL;	(* If true, the filter origin is shifted to the image center. *)
		fCutoffDistance	:	LREAL;	(* The cutoff distance of the Gaussian filter (> 0). *)
		fBandWidth	:	LREAL;	(* The band width of the Gaussian filter (> 0). *)
		hrPrev	:	HRESULT;	(* HRESULT indicating the result of previous operations (If SUCCEEDED(hrPrev) equals false, no operation is executed.) *)
	END_VAR

END_FUNCTION

// Functions/Fourier Analysis/F_VN_CreateBandrejectButterworthFilter

	{attribute 'TcIecLibraryType'}
	{attribute 'external_name' := 'F_VN_CreateBandrejectButterworthFilter_GUID_C41DA747_3CAD_4917_CB2F_3C02336F951C'}
	(* Creates a bandreject Butterworth filter, which can be applied to a frequency domain image by element-wise multiplication. *)
	FUNCTION F_VN_CreateBandrejectButterworthFilter : HRESULT
	VAR_INPUT
		ipFilter	:	REFERENCE TO ITcVnImage;	(* Returns the created filter (1 channel of type REAL or LREAL, depending on bDoublePrecision. Non-zero interface pointers are reused.). *)
		nWidth	:	UDINT;	(* Filter width (even, >= 2, must match the width of the image it is applied to) *)
		nHeight	:	UDINT;	(* Filter height (even, >= 2, must match the height of the image it is applied to) *)
		bDoublePrecision	:	BOOL;	(* If true, the filter is generated with double precision (LREAL) instead of single precision (REAL). *)
		bOriginAtCenter	:	BOOL;	(* If true, the filter origin is shifted to the image center. *)
		fCutoffDistance	:	LREAL;	(* The cutoff distance of the Butterworth filter (> 0). *)
		fBandWidth	:	LREAL;	(* The band width of the Butterworth filter (> 0). *)
		nOrder	:	UDINT;	(* The order of the Butterworth filter (> 0). *)
		fScale	:	LREAL;	(* The scale factor of the Butterworth filter denominator term (> 0, e.g. 0.414 or 1.0). *)
		hrPrev	:	HRESULT;	(* HRESULT indicating the result of previous operations (If SUCCEEDED(hrPrev) equals false, no operation is executed.) *)
	END_VAR

END_FUNCTION

// Functions/Fourier Analysis/F_VN_CreateBandrejectGaussianFilter

	{attribute 'TcIecLibraryType'}
	{attribute 'external_name' := 'F_VN_CreateBandrejectGaussianFilter_GUID_AAE3A500_C210_4B27_DB4D_79879B41F3DF'}
	(* Creates a bandreject Gaussian filter, which can be applied to a frequency domain image by element-wise multiplication. *)
	FUNCTION F_VN_CreateBandrejectGaussianFilter : HRESULT
	VAR_INPUT
		ipFilter	:	REFERENCE TO ITcVnImage;	(* Returns the created filter (1 channel of type REAL or LREAL, depending on bDoublePrecision. Non-zero interface pointers are reused.). *)
		nWidth	:	UDINT;	(* Filter width (even, >= 2, must match the width of the image it is applied to) *)
		nHeight	:	UDINT;	(* Filter height (even, >= 2, must match the height of the image it is applied to) *)
		bDoublePrecision	:	BOOL;	(* If true, the filter is generated with double precision (LREAL) instead of single precision (REAL). *)
		bOriginAtCenter	:	BOOL;	(* If true, the filter origin is shifted to the image center. *)
		fCutoffDistance	:	LREAL;	(* The cutoff distance of the Gaussian filter (> 0). *)
		fBandWidth	:	LREAL;	(* The band width of the Gaussian filter (> 0). *)
		hrPrev	:	HRESULT;	(* HRESULT indicating the result of previous operations (If SUCCEEDED(hrPrev) equals false, no operation is executed.) *)
	END_VAR

END_FUNCTION

// Functions/Fourier Analysis/F_VN_CreateHighpassButterworthFilter

	{attribute 'TcIecLibraryType'}
	{attribute 'external_name' := 'F_VN_CreateHighpassButterworthFilter_GUID_A1D1F13A_C2A9_4573_CCD1_D1D9C7E2C0B4'}
	(* Creates a highpass Butterworth filter, which can be applied to a frequency domain image by element-wise multiplication. *)
	FUNCTION F_VN_CreateHighpassButterworthFilter : HRESULT
	VAR_INPUT
		ipFilter	:	REFERENCE TO ITcVnImage;	(* Returns the created filter (1 channel of type REAL or LREAL, depending on bDoublePrecision. Non-zero interface pointers are reused.). *)
		nWidth	:	UDINT;	(* Filter width (even, >= 2, must match the width of the image it is applied to) *)
		nHeight	:	UDINT;	(* Filter height (even, >= 2, must match the height of the image it is applied to) *)
		bDoublePrecision	:	BOOL;	(* If true, the filter is generated with double precision (LREAL) instead of single precision (REAL). *)
		bOriginAtCenter	:	BOOL;	(* If true, the filter origin is shifted to the image center. *)
		fCutoffDistance	:	LREAL;	(* The cutoff distance of the Butterworth filter (> 0). *)
		nOrder	:	UDINT;	(* The order of the Butterworth filter (> 0). *)
		fScale	:	LREAL;	(* The scale factor of the Butterworth filter denominator term (> 0, e.g. 0.414 or 1.0). *)
		hrPrev	:	HRESULT;	(* HRESULT indicating the result of previous operations (If SUCCEEDED(hrPrev) equals false, no operation is executed.) *)
	END_VAR

END_FUNCTION

// Functions/Fourier Analysis/F_VN_CreateHighpassGaussianFilter

	{attribute 'TcIecLibraryType'}
	{attribute 'external_name' := 'F_VN_CreateHighpassGaussianFilter_GUID_16556F1B_488A_497E_ED81_F5E0BDC05145'}
	(* Creates a highpass Gaussian filter, which can be applied to a frequency domain image by element-wise multiplication. *)
	FUNCTION F_VN_CreateHighpassGaussianFilter : HRESULT
	VAR_INPUT
		ipFilter	:	REFERENCE TO ITcVnImage;	(* Returns the created filter (1 channel of type REAL or LREAL, depending on bDoublePrecision. Non-zero interface pointers are reused.). *)
		nWidth	:	UDINT;	(* Filter width (even, >= 2, must match the width of the image it is applied to) *)
		nHeight	:	UDINT;	(* Filter height (even, >= 2, must match the height of the image it is applied to) *)
		bDoublePrecision	:	BOOL;	(* If true, the filter is generated with double precision (LREAL) instead of single precision (REAL). *)
		bOriginAtCenter	:	BOOL;	(* If true, the filter origin is shifted to the image center. *)
		fCutoffDistance	:	LREAL;	(* The cutoff distance of the Gaussian filter (> 0). *)
		hrPrev	:	HRESULT;	(* HRESULT indicating the result of previous operations (If SUCCEEDED(hrPrev) equals false, no operation is executed.) *)
	END_VAR

END_FUNCTION

// Functions/Fourier Analysis/F_VN_CreateLowpassButterworthFilter

	{attribute 'TcIecLibraryType'}
	{attribute 'external_name' := 'F_VN_CreateLowpassButterworthFilter_GUID_B0D03C73_9889_4E08_C0AB_0EDD82A6EB9A'}
	(* Creates a lowpass Butterworth filter, which can be applied to a frequency domain image by element-wise multiplication. *)
	FUNCTION F_VN_CreateLowpassButterworthFilter : HRESULT
	VAR_INPUT
		ipFilter	:	REFERENCE TO ITcVnImage;	(* Returns the created filter (1 channel of type REAL or LREAL, depending on bDoublePrecision. Non-zero interface pointers are reused.). *)
		nWidth	:	UDINT;	(* Filter width (even, >= 2, must match the width of the image it is applied to) *)
		nHeight	:	UDINT;	(* Filter height (even, >= 2, must match the height of the image it is applied to) *)
		bDoublePrecision	:	BOOL;	(* If true, the filter is generated with double precision (LREAL) instead of single precision (REAL). *)
		bOriginAtCenter	:	BOOL;	(* If true, the filter origin is shifted to the image center. *)
		fCutoffDistance	:	LREAL;	(* The cutoff distance of the Butterworth filter (> 0). *)
		nOrder	:	UDINT;	(* The order of the Butterworth filter (> 0). *)
		fScale	:	LREAL;	(* The scale factor of the Butterworth filter denominator term (> 0, e.g. 0.414 or 1.0). *)
		hrPrev	:	HRESULT;	(* HRESULT indicating the result of previous operations (If SUCCEEDED(hrPrev) equals false, no operation is executed.) *)
	END_VAR

END_FUNCTION

// Functions/Fourier Analysis/F_VN_CreateLowpassGaussianFilter

	{attribute 'TcIecLibraryType'}
	{attribute 'external_name' := 'F_VN_CreateLowpassGaussianFilter_GUID_7BD6F64F_A61C_4033_E3C3_EA01FBB7F984'}
	(* Creates a lowpass Gaussian filter, which can be applied to a frequency domain image by element-wise multiplication. *)
	FUNCTION F_VN_CreateLowpassGaussianFilter : HRESULT
	VAR_INPUT
		ipFilter	:	REFERENCE TO ITcVnImage;	(* Returns the created filter (1 channel of type REAL or LREAL, depending on bDoublePrecision. Non-zero interface pointers are reused.). *)
		nWidth	:	UDINT;	(* Filter width (even, >= 2, must match the width of the image it is applied to) *)
		nHeight	:	UDINT;	(* Filter height (even, >= 2, must match the height of the image it is applied to) *)
		bDoublePrecision	:	BOOL;	(* If true, the filter is generated with double precision (LREAL) instead of single precision (REAL). *)
		bOriginAtCenter	:	BOOL;	(* If true, the filter origin is shifted to the image center. *)
		fCutoffDistance	:	LREAL;	(* The cutoff distance of the Gaussian filter (> 0). *)
		hrPrev	:	HRESULT;	(* HRESULT indicating the result of previous operations (If SUCCEEDED(hrPrev) equals false, no operation is executed.) *)
	END_VAR

END_FUNCTION

// Functions/Fourier Analysis/F_VN_Dft

	{attribute 'TcIecLibraryType'}
	{attribute 'external_name' := 'F_VN_Dft_GUID_1B32494D_248A_420A_E5A9_4369C71BE47B'}
	(* Computes the DFT for a given image. *)
	FUNCTION F_VN_Dft : HRESULT
	VAR_INPUT
		ipSpatialImage	:	ITcVnImage;	(* Source image (elements of type REAL or LREAL, 1 (Re) or 2 (Re + Im) channels) *)
		ipFrequencyImage	:	REFERENCE TO ITcVnImage;	(* Destination image (same type as ipSpatialImage, but number of channels and size can vary depending on bPackedCCS and bAutoPadding. *)
		bPackedCCS	:	BOOL;	(* If true and ipSpatialImage has only 1 channel, the result image will have 1 channel with packed complex-conjugate-symmetrical format results. Otherwise, the result image will have 2 separate channels (Re + Im), containing the full spectrum. *)
		bAutoPadding	:	BOOL;	(* If true, the input image is automatically padded (with 0s) to optimal size if required, to speed up dft (Creates a temporary copy so that ipSpatialImage content stays unchanged, which also requires some additional computation power. Therefore, it is recommended to compare execution times with and without padding.) *)
		hrPrev	:	HRESULT;	(* HRESULT indicating the result of previous operations (If SUCCEEDED(hrPrev) equals false, no operation is executed.) *)
	END_VAR

END_FUNCTION

// Functions/Fourier Analysis/F_VN_InverseDft

	{attribute 'TcIecLibraryType'}
	{attribute 'external_name' := 'F_VN_InverseDft_GUID_D6706B75_990D_43B1_C457_DBFD698F53C9'}
	(* Compute the inverse DFT for a given frequency image. *)
	FUNCTION F_VN_InverseDft : HRESULT
	VAR_INPUT
		ipFrequencyImage	:	ITcVnImage;	(* Source frequency image (elements of type REAL or LREAL, 1 (packed CCS) or 2 (Re + Im) channels) *)
		ipSpatialImage	:	REFERENCE TO ITcVnImage;	(* Destination image (Same type as ipFrequencyImage, but number of channels can vary depending on bRealOutput. An appropriate image will be created if required.) *)
		bRealOutput	:	BOOL;	(* Only relevant if ipFrequencyImage has 2 channels. If true, the result image will have only 1 channel. Otherwise, the result image will have 2 separate channels (Re + Im). If ipFrequencyImage has only 1 channel, packed CCS format is assumed and the result image will always have only 1 channel. *)
		hrPrev	:	HRESULT;	(* HRESULT indicating the result of previous operations (If SUCCEEDED(hrPrev) equals false, no operation is executed.) *)
	END_VAR

END_FUNCTION

// Functions/Fourier Analysis/F_VN_OptimalDftSize

	{attribute 'TcIecLibraryType'}
	{attribute 'external_name' := 'F_VN_OptimalDftSize_GUID_F8920499_45B0_4D40_FE9D_10C8C47031DD'}
	(* Computes the optimal image size for applying a dft (can lead to better performance). *)
	FUNCTION F_VN_OptimalDftSize : HRESULT
	VAR_INPUT
		ipImage	:	ITcVnImage;	(* Source image for which to compute the optimal width and height *)
	END_VAR
	VAR_IN_OUT
		nOptWidth	:	UDINT;	(* Returns the optimal width of the image *)
		nOptHeight	:	UDINT;	(* Returns the optimal height of the image *)
	END_VAR
	VAR_INPUT
		hrPrev	:	HRESULT;	(* HRESULT indicating the result of previous operations (If SUCCEEDED(hrPrev) equals false, no operation is executed.) *)
	END_VAR

END_FUNCTION

// Functions/Fourier Analysis/F_VN_PadImageBorder

	{attribute 'TcIecLibraryType'}
	{attribute 'external_name' := 'F_VN_PadImageBorder_GUID_852FCD40_BDFB_409A_C27C_BE0BB8D84FC2'}
	(* Add padding (zeros) around the original image borders. *)
	FUNCTION F_VN_PadImageBorder : HRESULT
	VAR_INPUT
		ipSrcImage	:	ITcVnImage;	(* Source image *)
		ipPaddedImage	:	REFERENCE TO ITcVnImage;	(* Padded destination image (Same type as ipSrcImage, an appropriate destination image will be created if required.) *)
		nTopBorder	:	UDINT;	(* Padding height in pixels above top border *)
		nBottomBorder	:	UDINT;	(* Padding height in pixels below bottom border *)
		nLeftBorder	:	UDINT;	(* Padding width in pixels before left border *)
		nRightBorder	:	UDINT;	(* Padding width in pixels after right border *)
		hrPrev	:	HRESULT;	(* HRESULT indicating the result of previous operations (If SUCCEEDED(hrPrev) equals false, no operation is executed.) *)
	END_VAR

END_FUNCTION

// Functions/Fourier Analysis/F_VN_PadImageBorderExp

	{attribute 'TcIecLibraryType'}
	{attribute 'external_name' := 'F_VN_PadImageBorderExp_GUID_22057AF7_8B4E_45BD_C0BE_4D1C001A3D6F'}
	(* Add padding around the original image borders. (expert function) *)
	FUNCTION F_VN_PadImageBorderExp : HRESULT
	VAR_INPUT
		ipSrcImage	:	ITcVnImage;	(* Source image *)
		ipPaddedImage	:	REFERENCE TO ITcVnImage;	(* Padded destination image (Same type as ipSrcImage, an appropriate destination image will be created if required.) *)
		nTopBorder	:	UDINT;	(* Padding height in pixels above top border *)
		nBottomBorder	:	UDINT;	(* Padding height in pixels below bottom border *)
		nLeftBorder	:	UDINT;	(* Padding width in pixels before left border *)
		nRightBorder	:	UDINT;	(* Padding width in pixels after right border *)
		ePaddingType	:	ETcVnBorderInterpolationMethod;	(* Specifies how the pixel values of the padding area are determined *)
	END_VAR
	VAR_IN_OUT
		aPaddingValue	:	TcVnVector4_LREAL;	(* Specifies the padding value if CONSTANT is used *)
	END_VAR
	VAR_INPUT
		hrPrev	:	HRESULT;	(* HRESULT indicating the result of previous operations (If SUCCEEDED(hrPrev) equals false, no operation is executed.) *)
	END_VAR

END_FUNCTION

// Functions/Machine Learning/F_VN_CreateBoostClassifier

	{attribute 'TcIecLibraryType'}
	{attribute 'external_name' := 'F_VN_CreateBoostClassifier_GUID_5975C274_601B_4843_C681_FA3F4BD9D3BE'}
	(* Create a Boost classifier using the default parameters. The initial reference count is set to one if a new model is created and kept, otherwise. The Boost classifier is only applicable to binary classification problems. It learns to distinguish between samples labelled with two user-defined class labels by incrementally adding weak classifiers to improve the classification results. Models of this type neither support on-line training (sample by sample) nor retraining. *)
	FUNCTION F_VN_CreateBoostClassifier : HRESULT
	VAR_INPUT
		ipMlModel	:	REFERENCE TO ITcVnMlModel;	(* Returns the created model (Non-zero interface pointers are reused.) *)
		hrPrev	:	HRESULT;	(* HRESULT indicating the result of previous operations (If SUCCEEDED(hrPrev) equals false, no operation is executed.) *)
	END_VAR

END_FUNCTION

// Functions/Machine Learning/F_VN_CreateBoostClassifierExp

	{attribute 'TcIecLibraryType'}
	{attribute 'external_name' := 'F_VN_CreateBoostClassifierExp_GUID_5C507CCA_8178_40E6_D313_30A20CA7691E'}
	(* Create a Boost classifier. The initial reference count is set to one if a new model is created and kept, otherwise. The Boost classifier is only applicable to binary classification problems. It learns to distinguish between samples labelled with two user-defined class labels by incrementally adding weak classifiers to improve the classification results. Models of this type neither support on-line training (sample by sample) nor retraining. (expert function) *)
	FUNCTION F_VN_CreateBoostClassifierExp : HRESULT
	VAR_INPUT
		ipMlModel	:	REFERENCE TO ITcVnMlModel;	(* Returns the created model (Non-zero interface pointers are reused.) *)
		eType	:	ETcVnBoostClassifierType;	(* Learning algorithm type (default: TCVN_BCT_REAL) *)
		nMaxDepth	:	UDINT;	(* Maximum tree depth (default: 1) *)
		nMinSamples	:	UDINT;	(* Minimum number of samples within a node required for splitting (default: 10) *)
		nWeakClassifiers	:	UDINT;	(* Number of weak classifiers (default: 100) *)
		fWeightTrimRate	:	LREAL;	(* Weight threshold used during training (off: 0; default: 0.95). *)
		hrPrev	:	HRESULT;	(* HRESULT indicating the result of previous operations (If SUCCEEDED(hrPrev) equals false, no operation is executed.) *)
	END_VAR

END_FUNCTION

// Functions/Machine Learning/F_VN_CreateBoostClassifierExp2

	{attribute 'TcIecLibraryType'}
	{attribute 'external_name' := 'F_VN_CreateBoostClassifierExp2_GUID_E84F016B_6A31_4FFB_C157_738998FA28C1'}
	(* Create a Boost classifier. The initial reference count is set to one if a new model is created and kept, otherwise. The Boost classifier is only applicable to binary classification problems. It learns to distinguish between samples labelled with two user-defined class labels by incrementally adding weak classifiers to improve the classification results. Models of this type neither support on-line training (sample by sample) nor retraining. (expert function) *)
	FUNCTION F_VN_CreateBoostClassifierExp2 : HRESULT
	VAR_INPUT
		ipMlModel	:	REFERENCE TO ITcVnMlModel;	(* Returns the created model (Non-zero interface pointers are reused.) *)
		eType	:	ETcVnBoostClassifierType;	(* Learning algorithm type (default: TCVN_BCT_REAL) *)
		nMaxDepth	:	UDINT;	(* Maximum tree depth (default: 1) *)
		nMinSamples	:	UDINT;	(* Minimum number of samples within a node required for splitting (default: 10) *)
		nWeakClassifiers	:	UDINT;	(* Number of weak classifiers (default: 100) *)
		fWeightTrimRate	:	LREAL;	(* Weight threshold used during training (off: 0; default: 0.95). *)
		ipClassPriors	:	ITcVnContainer;	(* Class priors (ContainerType_Vector_REAL or ContainerType_Vector_LREAL; only for classifiers; optional, set to 0 if not required or not allowed; default: 0) *)
		hrPrev	:	HRESULT;	(* HRESULT indicating the result of previous operations (If SUCCEEDED(hrPrev) equals false, no operation is executed.) *)
	END_VAR

END_FUNCTION

// Functions/Machine Learning/F_VN_CreateKmppModel

	{attribute 'TcIecLibraryType'}
	{attribute 'external_name' := 'F_VN_CreateKmppModel_GUID_7BD1738D_4999_47CE_FC07_4F434267295B'}
	(* Create a k-means++ model of the specified type. The initial reference count is set to one if a new model is created and kept, otherwise. Models of this type neither support on-line training (sample by sample) nor retraining. *)
	FUNCTION F_VN_CreateKmppModel : HRESULT
	VAR_INPUT
		ipMlModel	:	REFERENCE TO ITcVnMlModel;	(* Returns the created model (Non-zero interface pointers are reused.) *)
		eKmppType	:	ETcVnPrototypeClusterer;	(* k-means++ model type *)
		nK	:	UDINT;	(* Parameter k (number of clusters) *)
		hrPrev	:	HRESULT;	(* HRESULT indicating the result of previous operations (If SUCCEEDED(hrPrev) equals false, no operation is executed.) *)
	END_VAR

END_FUNCTION

// Functions/Machine Learning/F_VN_CreateKmppModelExp

	{attribute 'TcIecLibraryType'}
	{attribute 'external_name' := 'F_VN_CreateKmppModelExp_GUID_1687B1AB_AD3B_48ED_D77C_DB76DC86EB53'}
	(* Create a k-means++ model of the specified type. The initial reference count is set to one if a new model is created and kept, otherwise. Models of this type neither support on-line training (sample by sample) nor retraining. (expert function) *)
	FUNCTION F_VN_CreateKmppModelExp : HRESULT
	VAR_INPUT
		ipMlModel	:	REFERENCE TO ITcVnMlModel;	(* Returns the created model (Non-zero interface pointers are reused.) *)
		eKmppType	:	ETcVnPrototypeClusterer;	(* k-means++ model type *)
		nK	:	UDINT;	(* Parameter k (number of clusters) *)
		bDoublePrecision	:	BOOL;	(* If true, the model is generated with double precision (LREAL) instead of single precision (REAL). (default: FALSE) *)
		nMaxIterations	:	UDINT;	(* Maximum number of iterations (triggers the usage of the default value of 10 if it equals 0) *)
		fEpsilon	:	LREAL;	(* Maximum allowed difference of the error between two successive iterations (triggers the usage of the default value of 0.001 if it equals 0) *)
		hrPrev	:	HRESULT;	(* HRESULT indicating the result of previous operations (If SUCCEEDED(hrPrev) equals false, no operation is executed.) *)
	END_VAR

END_FUNCTION

// Functions/Machine Learning/F_VN_CreateKnnModel

	{attribute 'TcIecLibraryType'}
	{attribute 'external_name' := 'F_VN_CreateKnnModel_GUID_B8250D66_8EC6_4BF2_D6D9_76FBC4F3DC13'}
	(* Create a k-nearest neighbors model of the specified type. The initial reference count is set to one if a new model is created and kept, otherwise. Models of this type support on-line training (sample by sample) and retraining. Predictions can only be scalar. *)
	FUNCTION F_VN_CreateKnnModel : HRESULT
	VAR_INPUT
		ipMlModel	:	REFERENCE TO ITcVnMlModel;	(* Returns the created model (Non-zero interface pointers are reused.) *)
		eKnnType	:	ETcVnKnn;	(* k-nearest neighbors model type *)
		nK	:	UDINT;	(* Parameter k used for prediction (number of considered neighbors) *)
		hrPrev	:	HRESULT;	(* HRESULT indicating the result of previous operations (If SUCCEEDED(hrPrev) equals false, no operation is executed.) *)
	END_VAR

END_FUNCTION

// Functions/Machine Learning/F_VN_CreateLbgModel

	{attribute 'TcIecLibraryType'}
	{attribute 'external_name' := 'F_VN_CreateLbgModel_GUID_2F7FBCED_94CF_4926_CDCB_E3CB8F150CAB'}
	(* Create a LBG model of the specified type. The initial reference count is set to one if a new model is created and kept, otherwise. Models of this type neither support on-line training (sample by sample) nor retraining. *)
	FUNCTION F_VN_CreateLbgModel : HRESULT
	VAR_INPUT
		ipMlModel	:	REFERENCE TO ITcVnMlModel;	(* Returns the created model (Non-zero interface pointers are reused.) *)
		eLbgType	:	ETcVnPrototypeClusterer;	(* LBG model type *)
		nMaxClusters	:	UDINT;	(* Maximum number of clusters *)
		fMaxClusterRadius	:	LREAL;	(* Maximum allowed radius (L2 norm) of a single cluster, i.e. clusters with a higher radius will be split into smaller ones, until a global number of nMaxClusters is reached. *)
		bSingleSplitSteps	:	BOOL;	(* If true, the global optimization is always run after a single cluster has been split. If false, several clusters are split within the same step before applying the global optimization. Applying the global optimization less often is faster, but can lead to less optimal results, especially having 2 nearby clusters that could be represented by 1. *)
		hrPrev	:	HRESULT;	(* HRESULT indicating the result of previous operations (If SUCCEEDED(hrPrev) equals false, no operation is executed.) *)
	END_VAR

END_FUNCTION

// Functions/Machine Learning/F_VN_CreateLbgModelExp

	{attribute 'TcIecLibraryType'}
	{attribute 'external_name' := 'F_VN_CreateLbgModelExp_GUID_FA609D9D_F94C_48E6_F186_ECEECAAE11ED'}
	(* Create a LBG model of the specified type. The initial reference count is set to one if a new model is created and kept, otherwise. Models of this type neither support on-line training (sample by sample) nor retraining. (expert function) *)
	FUNCTION F_VN_CreateLbgModelExp : HRESULT
	VAR_INPUT
		ipMlModel	:	REFERENCE TO ITcVnMlModel;	(* Returns the created model (Non-zero interface pointers are reused.) *)
		eLbgType	:	ETcVnPrototypeClusterer;	(* LBG model type *)
		nMaxClusters	:	UDINT;	(* Maximum number of clusters *)
		fMaxClusterRadius	:	LREAL;	(* Maximum allowed radius (L2 norm) of a single cluster, i.e. clusters with a higher radius will be split into smaller ones, until a global number of nMaxClusters is reached. *)
		bSingleSplitSteps	:	BOOL;	(* If true, the global optimization is always run after a single cluster has been split. If false, several clusters are split within the same step before applying the global optimization. Applying the global optimization less often is faster, but can lead to less optimal results, especially having 2 nearby clusters that could be represented by 1. *)
		bDoublePrecision	:	BOOL;	(* If true, the model is generated with double precision (LREAL) instead of single precision (REAL). (default: FALSE) *)
		nMaxIterations	:	UDINT;	(* Maximum number of iterations (triggers the usage of the default value of 10 if it equals 0) *)
		fEpsilon	:	LREAL;	(* Maximum allowed difference of the error between two successive iterations (triggers the usage of the default value of 0.001 if it equals 0) *)
		hrPrev	:	HRESULT;	(* HRESULT indicating the result of previous operations (If SUCCEEDED(hrPrev) equals false, no operation is executed.) *)
	END_VAR

END_FUNCTION

// Functions/Machine Learning/F_VN_CreateLdaTransform

	{attribute 'TcIecLibraryType'}
	{attribute 'external_name' := 'F_VN_CreateLdaTransform_GUID_380EC1B5_80F2_40D8_CEFD_064E18452A47'}
	(* Create an LDA-based feature transform from the provided data. The number of samples must be >= the number of features and the number of classes must be >= 2. The initial reference count is set to one if a new model is created and kept, otherwise. *)
	FUNCTION F_VN_CreateLdaTransform : HRESULT
	VAR_INPUT
		ipMlModel	:	REFERENCE TO ITcVnMlModel;	(* Returns the created feature transform (Non-zero interface pointers are reused.) *)
		ipSamples	:	ITcUnknown;	(* Container holding a batch of input samples (ContainerType_Vector_Vector_REAL or ContainerType_Vector_Vector_LREAL) *)
		ipClasses	:	ITcVnContainer;	(* Class labels corresponding to the input samples (ContainerType_Vector_DINT) *)
		hrPrev	:	HRESULT;	(* HRESULT indicating the result of previous operations (If SUCCEEDED(hrPrev) equals false, no operation is executed.) *)
	END_VAR

END_FUNCTION

// Functions/Machine Learning/F_VN_CreateLdaTransformViaComponentNum

	{attribute 'TcIecLibraryType'}
	{attribute 'external_name' := 'F_VN_CreateLdaTransformViaComponentNum_GUID_1C0AEC56_8E94_4D96_DA16_997B250C98FA'}
	(* Create an LDA-based feature transform from the provided data where the number of components to be used is predefined. The number of samples must be >= the number of features and the number of classes must be >= 2. The initial reference count is set to one if a new model is created and kept, otherwise. (expert function) *)
	FUNCTION F_VN_CreateLdaTransformViaComponentNum : HRESULT
	VAR_INPUT
		ipMlModel	:	REFERENCE TO ITcVnMlModel;	(* Returns the created feature transform (Non-zero interface pointers are reused.) *)
		ipSamples	:	ITcUnknown;	(* Container holding a batch of input samples (ContainerType_Vector_Vector_REAL or ContainerType_Vector_Vector_LREAL) *)
		ipClasses	:	ITcVnContainer;	(* Class labels corresponding to the input samples (ContainerType_Vector_DINT) *)
		nComponentNum	:	UDINT;	(* Number of components (nComponentNum must be smaller than the number of classes. A value of 0 results in the automatic computation of the maximum number of components.) *)
		hrPrev	:	HRESULT;	(* HRESULT indicating the result of previous operations (If SUCCEEDED(hrPrev) equals false, no operation is executed.) *)
	END_VAR

END_FUNCTION

// Functions/Machine Learning/F_VN_CreateNbcModel

	{attribute 'TcIecLibraryType'}
	{attribute 'external_name' := 'F_VN_CreateNbcModel_GUID_5DE26C09_929C_485C_DF79_BFA65B0752BE'}
	(* Create a normal Bayes classifier of the specified type. The initial reference count is set to one if a new model is created and kept, otherwise. In order to train normal Bayes classifiers, a sufficiently high number of samples is required for each class. It depends on the number of features and the distribution of the data. Hence, it needs to be tested for each application. Models of this type do not support on-line training (sample by sample). For the retraining of such classifier models, the set of presented classes must be identical to the previous learning steps. Otherwise, an exception is raised. *)
	FUNCTION F_VN_CreateNbcModel : HRESULT
	VAR_INPUT
		ipMlModel	:	REFERENCE TO ITcVnMlModel;	(* Returns the created model (Non-zero interface pointers are reused.) *)
		eNbcType	:	ETcVnNbc;	(* Normal Bayes classifier type *)
		hrPrev	:	HRESULT;	(* HRESULT indicating the result of previous operations (If SUCCEEDED(hrPrev) equals false, no operation is executed.) *)
	END_VAR

END_FUNCTION

// Functions/Machine Learning/F_VN_CreatePcaTransform

	{attribute 'TcIecLibraryType'}
	{attribute 'external_name' := 'F_VN_CreatePcaTransform_GUID_5DC46F49_5969_4771_E91D_37F977C0E078'}
	(* Create a PCA-based feature transform from the provided data. The maximum number of principal components that can be computed equals the minimum of the number of samples and the number of features. The initial reference count is set to one if a new model is created and kept, otherwise. *)
	FUNCTION F_VN_CreatePcaTransform : HRESULT
	VAR_INPUT
		ipMlModel	:	REFERENCE TO ITcVnMlModel;	(* Returns the created feature transform (Non-zero interface pointers are reused.) *)
		ipSamples	:	ITcUnknown;	(* Container holding a batch of input samples (ContainerType_Vector_Vector_REAL or ContainerType_Vector_Vector_LREAL) *)
		hrPrev	:	HRESULT;	(* HRESULT indicating the result of previous operations (If SUCCEEDED(hrPrev) equals false, no operation is executed.) *)
	END_VAR

END_FUNCTION

// Functions/Machine Learning/F_VN_CreatePcaTransformViaComponentNum

	{attribute 'TcIecLibraryType'}
	{attribute 'external_name' := 'F_VN_CreatePcaTransformViaComponentNum_GUID_AFF0E4E0_F744_4858_FE7C_4EC2816DEE62'}
	(* Create a PCA-based feature transform from the provided data where the number of prinicpal components to be used is predefined. The maximum number of principal components that can be computed equals the minimum of the number of samples and the number of features. The initial reference count is set to one if a new model is created and kept, otherwise. (expert function) *)
	FUNCTION F_VN_CreatePcaTransformViaComponentNum : HRESULT
	VAR_INPUT
		ipMlModel	:	REFERENCE TO ITcVnMlModel;	(* Returns the created feature transform (Non-zero interface pointers are reused.) *)
		ipSamples	:	ITcUnknown;	(* Container holding a batch of input samples (ContainerType_Vector_Vector_REAL or ContainerType_Vector_Vector_LREAL) *)
		nComponentNum	:	UDINT;	(* Number of principal components (A value of 0 results in the automatic computation of the maximum number of components.) *)
		hrPrev	:	HRESULT;	(* HRESULT indicating the result of previous operations (If SUCCEEDED(hrPrev) equals false, no operation is executed.) *)
	END_VAR

END_FUNCTION

// Functions/Machine Learning/F_VN_CreatePcaTransformViaVariance

	{attribute 'TcIecLibraryType'}
	{attribute 'external_name' := 'F_VN_CreatePcaTransformViaVariance_GUID_9AE01371_A920_4CFF_D3A7_B6D63F1D7982'}
	(* Create a PCA-based feature transform from the provided data based on a given fraction of variance to be retained. The maximum number of principal components that can be computed equals the minimum of the number of samples and the number of features. The initial reference count is set to one if a new model is created and kept, otherwise. (expert function) *)
	FUNCTION F_VN_CreatePcaTransformViaVariance : HRESULT
	VAR_INPUT
		ipMlModel	:	REFERENCE TO ITcVnMlModel;	(* Returns the created feature transform (Non-zero interface pointers are reused.) *)
		ipSamples	:	ITcUnknown;	(* Container holding a batch of input samples (ContainerType_Vector_Vector_REAL or ContainerType_Vector_Vector_LREAL) *)
		fRetainedVariance	:	LREAL;	(* Fraction of variance that is to be retained by the PCA (A value of 1.0 signifies 100%.) *)
		hrPrev	:	HRESULT;	(* HRESULT indicating the result of previous operations (If SUCCEEDED(hrPrev) equals false, no operation is executed.) *)
	END_VAR

END_FUNCTION

// Functions/Machine Learning/F_VN_CreateRTreesModel

	{attribute 'TcIecLibraryType'}
	{attribute 'external_name' := 'F_VN_CreateRTreesModel_GUID_D96DB75E_CA94_4473_F3AF_32D380CE7973'}
	(* Create a random trees model of the specified type. The initial reference count is set to one if a new model is created and kept, otherwise. Models of this type neither support on-line training (sample by sample) nor retraining. Predictions can only be scalar. *)
	FUNCTION F_VN_CreateRTreesModel : HRESULT
	VAR_INPUT
		ipMlModel	:	REFERENCE TO ITcVnMlModel;	(* Returns the created model (Non-zero interface pointers are reused.) *)
		eRTreesType	:	ETcVnRTrees;	(* Random trees model type *)
		hrPrev	:	HRESULT;	(* HRESULT indicating the result of previous operations (If SUCCEEDED(hrPrev) equals false, no operation is executed.) *)
	END_VAR

END_FUNCTION

// Functions/Machine Learning/F_VN_CreateRTreesModelExp

	{attribute 'TcIecLibraryType'}
	{attribute 'external_name' := 'F_VN_CreateRTreesModelExp_GUID_33D995F5_FF65_4811_C7AE_0DAADF41F415'}
	(* Create a random trees model of the specified type. The initial reference count is set to one if a new model is created and kept, otherwise. Models of this type neither support on-line training (sample by sample) nor retraining. Predictions can only be scalar. (expert function) *)
	FUNCTION F_VN_CreateRTreesModelExp : HRESULT
	VAR_INPUT
		ipMlModel	:	REFERENCE TO ITcVnMlModel;	(* Returns the created model (Non-zero interface pointers are reused.) *)
		eRTreesType	:	ETcVnRTrees;	(* Random trees model type *)
		nMaxDepth	:	UDINT;	(* Maximum tree depth (default: 5) *)
		nMinSamples	:	UDINT;	(* Minimum number of samples within a node required for splitting (default: 10) *)
		nActiveVariables	:	UDINT;	(* Number of variables considered for splitting (0 means sqrt(total number of variables); default: 0) *)
		nMaxIterations	:	UDINT;	(* Maximum number of iterations (disabled if it equals 0 and fEpsilon is different from 0.0; triggers the usage of the default value of 50 if nMaxIterations and fEpsilon equal 0) *)
		fEpsilon	:	LREAL;	(* Maximum allowed difference of the error between two successive iterations (disabled if it equals 0.0 and nMaxIterations is different from 0; triggers the usage of the default value of 0.1 if nMaxIterations and fEpsilon equal 0) *)
		hrPrev	:	HRESULT;	(* HRESULT indicating the result of previous operations (If SUCCEEDED(hrPrev) equals false, no operation is executed.) *)
	END_VAR

END_FUNCTION

// Functions/Machine Learning/F_VN_CreateRTreesModelExp2

	{attribute 'TcIecLibraryType'}
	{attribute 'external_name' := 'F_VN_CreateRTreesModelExp2_GUID_4CCAAFB9_BCFA_49D3_DA45_0FED5B3DCEA9'}
	(* Create a random trees model of the specified type. The initial reference count is set to one if a new model is created and kept, otherwise. Models of this type neither support on-line training (sample by sample) nor retraining. Predictions can only be scalar. (expert function) *)
	FUNCTION F_VN_CreateRTreesModelExp2 : HRESULT
	VAR_INPUT
		ipMlModel	:	REFERENCE TO ITcVnMlModel;	(* Returns the created model (Non-zero interface pointers are reused.) *)
		eRTreesType	:	ETcVnRTrees;	(* Random trees model type *)
		nMaxDepth	:	UDINT;	(* Maximum tree depth (default: 5) *)
		nMinSamples	:	UDINT;	(* Minimum number of samples within a node required for splitting (default: 10) *)
		nActiveVariables	:	UDINT;	(* Number of variables considered for splitting (0 means sqrt(total number of variables); default: 0) *)
		nMaxIterations	:	UDINT;	(* Maximum number of iterations (disabled if it equals 0 and fEpsilon is different from 0.0; triggers the usage of the default value of 50 if nMaxIterations and fEpsilon equal 0) *)
		fEpsilon	:	LREAL;	(* Maximum allowed difference of the error between two successive iterations (disabled if it equals 0.0 and nMaxIterations is different from 0; triggers the usage of the default value of 0.1 if nMaxIterations and fEpsilon equal 0) *)
		fRegressionAccuracy	:	REAL;	(* Termination criterion for regressors (only for regressors; set to default if not allowed; default: 0.0) *)
		ipClassPriors	:	ITcVnContainer;	(* Class priors (ContainerType_Vector_REAL or ContainerType_Vector_LREAL; only for classifiers; optional, set to 0 if not required or not allowed; default: 0) *)
		hrPrev	:	HRESULT;	(* HRESULT indicating the result of previous operations (If SUCCEEDED(hrPrev) equals false, no operation is executed.) *)
	END_VAR

END_FUNCTION

// Functions/Machine Learning/F_VN_CreateStaModel

